	{attribute 'TcIecLibraryType'}
	{attribute 'external_name' := 'F_VN_CalibrateLinescanCameraExp_GUID_4678BC8A_FAF5_BD22_52B3_D89A3D1569BD'}
	(* Compute the camera parameters (intrinsic + extrinsic) by evaluating images containing a line calibration pattern. The pattern must consist of alternating vertical and diagonal lines, with each diagonal having the same constant slope: |\|\|...\|. The results are only valid for the x-direction of a line scan image. To get accurate x-values for a transformation into world coordinates, the y-coordinate must be set to half the sensor width and so equal to the cy-value of the camera matrix. For other y-values, the results are approximated and can be inaccurate. The extrinsic parameters are computed for the first image in the array. (expert function) *)
	FUNCTION F_VN_CalibrateLinescanCameraExp : HRESULT
	VAR_INPUT
		pSrcImages	:	PVOID;	(* Pointer to an array of 1 or more source images (1 channel). If the images have more than 1 row, each row must contain an image of the same pattern position. *)
		nSrcArraySize	:	UINT;	(* pSrcImages array size *)
		ipPatternLineOrigins	:	ITcVnContainer;	(* X position of the pattern line origins (ContainerType_Vector_REAL, usually same origin for vertical and following diagonal line) *)
		fSlopeRad	:	LREAL;	(* Slope of the diagonal line in rad (> 0, < PI/2), relative to the vertical line (i.e., 0 would be a vertical line, PI/2 a horizontal line) *)
	END_VAR
	VAR_IN_OUT
		aCameraMatrix	:	TcVnMatrix3x3_LREAL;	(* Returns the camera matrix *)
		aDistortionCoefficients	:	TcVnArray8_LREAL;	(* Returns the lens distortion coefficients [k1, k2, p1, p2, k3, k4, k5, k6] *)
		aRotationMatrix	:	TcVnMatrix3x3_LREAL;	(* Returns the rotation matrix *)
		aTranslationVector	:	TcVnVector3_LREAL;	(* Returns the translation vector *)
		fReprojError	:	LREAL;	(* Returns the reprojection error *)
		stCalibrationOptions	:	TcVnCameraCalibrationOptions;	(* Calibration options (recommended to set bFixAspectRatio, bFixPrincipalPoint, bZeroTangentDist) *)
	END_VAR
	VAR_INPUT
		eEdgeDirection	:	ETcVnEdgeDirection;	(* Specification of the edge direction to search for *)
		fMinStrength	:	REAL;	(* Specification of the minimum strength (intensity difference) of the edge to search for *)
		nMaxSearchLines	:	UDINT;	(* Maximum number of search lines (equally distributed over the image height, at most 1 searchline per image row) *)
		nMaxThickness	:	UDINT;	(* Specification of the maximum thickness of the edge to search for, which means fMinStrength must be reached within nMaxThickness pixels *)
		nSubpixelsIterations	:	UDINT;	(* Specifies the number of subpixels (for INTERPOLATION, 10 - 20 usually is sufficient) or maximum number of iterations for optimizing the parameters (for APPROX_ERF and APPROX_GAUSSIAN, 50 - 100 usually is sufficient) *)
		fApproxPrecision	:	REAL;	(* Specifies the approximation precision for APPROX_ERF and APPROX_GAUSSIAN (0.001 usually is sufficient, unused for INTERPOLATION) *)
		eAlgorithm	:	ETcVnEdgeDetectionAlgorithm;	(* Selection of the edge detection algorithm *)
		hrPrev	:	HRESULT;	(* HRESULT indicating the result of previous operations (If SUCCEEDED(hrPrev) equals false, no operation is executed.) *)
	END_VAR

END_FUNCTION

// Functions/Geometric and Coordinate Transformations/Calibration/F_VN_CompensateLensDistortion

	{attribute 'TcIecLibraryType'}
	{attribute 'external_name' := 'F_VN_CompensateLensDistortion_GUID_A3855505_9E36_B648_4D9A_72404444EE18'}
	(* Transforms an image to compensate the lens distortion. *)
	FUNCTION F_VN_CompensateLensDistortion : HRESULT
	VAR_INPUT
		ipSrcImage	:	ITcVnImage;	(* Source image *)
		ipDestImage	:	REFERENCE TO ITcVnImage;	(* Destination image (An appropriate destination image will be created if required.) *)
	END_VAR
	VAR_IN_OUT
		aCameraMatrix	:	TcVnMatrix3x3_LREAL;	(* Camera matrix containing the intrinsic parameters *)
		aDistortionCoefficients	:	TcVnArray4_LREAL;	(* Lens distortion coefficients [k1, k2, p1, p2] *)
	END_VAR
	VAR_INPUT
		hrPrev	:	HRESULT;	(* HRESULT indicating the result of previous operations (If SUCCEEDED(hrPrev) equals false, no operation is executed.) *)
	END_VAR

END_FUNCTION

// Functions/Geometric and Coordinate Transformations/Calibration/F_VN_CompensateLensDistortionExp1

	{attribute 'TcIecLibraryType'}
	{attribute 'external_name' := 'F_VN_CompensateLensDistortionExp1_GUID_39F83302_C215_BA53_4A0E_6585051CD298'}
	(* Transforms an image to compensate the lens distortion. (expert function) *)
	FUNCTION F_VN_CompensateLensDistortionExp1 : HRESULT
	VAR_INPUT
		ipSrcImage	:	ITcVnImage;	(* Source image *)
		ipDestImage	:	REFERENCE TO ITcVnImage;	(* Destination image (An appropriate destination image will be created if required.) *)
	END_VAR
	VAR_IN_OUT
		aCameraMatrix	:	TcVnMatrix3x3_LREAL;	(* Camera matrix containing the intrinsic parameters *)
		aDistortionCoefficients	:	TcVnArray8_LREAL;	(* Lens distortion coefficients [k1, k2, p1, p2, k3, k4, k5, k6] *)
	END_VAR
	VAR_INPUT
		hrPrev	:	HRESULT;	(* HRESULT indicating the result of previous operations (If SUCCEEDED(hrPrev) equals false, no operation is executed.) *)
	END_VAR

END_FUNCTION

// Functions/Geometric and Coordinate Transformations/Calibration/F_VN_CompensateLensDistortionExp2

	{attribute 'TcIecLibraryType'}
	{attribute 'external_name' := 'F_VN_CompensateLensDistortionExp2_GUID_C6636C8E_8710_BA51_6E0A_CA8278B52EE8'}
	(* Transforms an image to compensate the lens distortion. (expert function) *)
	FUNCTION F_VN_CompensateLensDistortionExp2 : HRESULT
	VAR_INPUT
		ipSrcImage	:	ITcVnImage;	(* Source image *)
		ipDestImage	:	REFERENCE TO ITcVnImage;	(* Destination image (An appropriate destination image will be created if required.) *)
	END_VAR
	VAR_IN_OUT
		aCameraMatrix	:	TcVnMatrix3x3_LREAL;	(* Camera matrix containing the intrinsic parameters *)
		aDistortionCoefficients	:	TcVnArray8_LREAL;	(* Lens distortion coefficients [k1, k2, p1, p2, k3, k4, k5, k6] *)
		aNewCameraMatrix	:	TcVnMatrix3x3_LREAL;	(* Allows additional scaling and shifting of the result image *)
	END_VAR
	VAR_INPUT
		hrPrev	:	HRESULT;	(* HRESULT indicating the result of previous operations (If SUCCEEDED(hrPrev) equals false, no operation is executed.) *)
	END_VAR

END_FUNCTION

// Functions/Geometric and Coordinate Transformations/Calibration/F_VN_CompensateLensDistortionForPoints

	{attribute 'TcIecLibraryType'}
	{attribute 'external_name' := 'F_VN_CompensateLensDistortionForPoints_GUID_1E1DEE69_79BC_BA65_762B_E597A5CC1182'}
	(* Transforms point coordinates to compensate the lens distortion. *)
	FUNCTION F_VN_CompensateLensDistortionForPoints : HRESULT
	VAR_INPUT
		ipSrcPoints	:	ITcVnContainer;	(* Container with source point coordinates (ContainerType_Vector_TcVnPoint2_REAL or ContainerType_Vector_TcVnPoint2_DINT) *)
		ipDestPoints	:	REFERENCE TO ITcVnContainer;	(* Returns a container with the transformed point coordinates (ContainerType_Vector_TcVnPoint2_REAL) *)
	END_VAR
	VAR_IN_OUT
		aCameraMatrix	:	TcVnMatrix3x3_LREAL;	(* Camera matrix containing the intrinsic parameters *)
		aDistortionCoefficients	:	TcVnArray4_LREAL;	(* Lens distortion coefficients [k1, k2, p1, p2] *)
	END_VAR
	VAR_INPUT
		hrPrev	:	HRESULT;	(* HRESULT indicating the result of previous operations (If SUCCEEDED(hrPrev) equals false, no operation is executed.) *)
	END_VAR

END_FUNCTION

// Functions/Geometric and Coordinate Transformations/Calibration/F_VN_CompensateLensDistortionForPointsExp1

	{attribute 'TcIecLibraryType'}
	{attribute 'external_name' := 'F_VN_CompensateLensDistortionForPointsExp1_GUID_7FE839DD_7A8B_BA4D_4709_CA0E7CDDBA0C'}
	(* Transforms point coordinates to compensate the lens distortion. (expert function) *)
	FUNCTION F_VN_CompensateLensDistortionForPointsExp1 : HRESULT
	VAR_INPUT
		ipSrcPoints	:	ITcVnContainer;	(* Container with source point coordinates (ContainerType_Vector_TcVnPoint2_REAL or ContainerType_Vector_TcVnPoint2_DINT) *)
		ipDestPoints	:	REFERENCE TO ITcVnContainer;	(* Returns a container with the transformed point coordinates (ContainerType_Vector_TcVnPoint2_REAL) *)
	END_VAR
	VAR_IN_OUT
		aCameraMatrix	:	TcVnMatrix3x3_LREAL;	(* Camera matrix containing the intrinsic parameters *)
		aDistortionCoefficients	:	TcVnArray8_LREAL;	(* Lens distortion coefficients [k1, k2, p1, p2, k3, k4, k5, k6] *)
	END_VAR
	VAR_INPUT
		hrPrev	:	HRESULT;	(* HRESULT indicating the result of previous operations (If SUCCEEDED(hrPrev) equals false, no operation is executed.) *)
	END_VAR

END_FUNCTION

// Functions/Geometric and Coordinate Transformations/Calibration/F_VN_CompensateLensDistortionForPointsExp2

	{attribute 'TcIecLibraryType'}
	{attribute 'external_name' := 'F_VN_CompensateLensDistortionForPointsExp2_GUID_30396D32_CFFC_B079_658D_44A89CF24BD9'}
	(* Transforms point coordinates to compensate the lens distortion. (expert function) *)
	FUNCTION F_VN_CompensateLensDistortionForPointsExp2 : HRESULT
	VAR_INPUT
		ipSrcPoints	:	ITcVnContainer;	(* Container with source point coordinates (ContainerType_Vector_TcVnPoint2_REAL or ContainerType_Vector_TcVnPoint2_DINT) *)
		ipDestPoints	:	REFERENCE TO ITcVnContainer;	(* Returns a container with the transformed point coordinates (ContainerType_Vector_TcVnPoint2_REAL) *)
	END_VAR
	VAR_IN_OUT
		aCameraMatrix	:	TcVnMatrix3x3_LREAL;	(* Camera matrix containing the intrinsic parameters *)
		aDistortionCoefficients	:	TcVnArray8_LREAL;	(* Lens distortion coefficients [k1, k2, p1, p2, k3, k4, k5, k6] *)
		aNewCameraMatrix	:	TcVnMatrix3x3_LREAL;	(* Allows additional shifting of the result point coordinates *)
	END_VAR
	VAR_INPUT
		hrPrev	:	HRESULT;	(* HRESULT indicating the result of previous operations (If SUCCEEDED(hrPrev) equals false, no operation is executed.) *)
	END_VAR

END_FUNCTION

// Functions/Geometric and Coordinate Transformations/Calibration/F_VN_DetectPatternPoints

	{attribute 'TcIecLibraryType'}
	{attribute 'external_name' := 'F_VN_DetectPatternPoints_GUID_E5D619D4_AB2C_BCDF_69FA_59048593E7EE'}
	(* Detects calibration pattern points (circles) within the provided image. *)
	FUNCTION F_VN_DetectPatternPoints : HRESULT
	VAR_INPUT
		ipSrcImage	:	ITcVnImage;	(* Source image (USINT, 1 channel) *)
		ipPatternPoints	:	REFERENCE TO ITcVnContainer;	(* Returns the pattern point positions (ContainerType_Vector_TcVnPoint2_REAL; Non-zero interface pointers are reused.) *)
	END_VAR
	VAR_IN_OUT
		stBlobDetectionParams	:	TcVnParamsBlobDetection;	(* Parameters to detect and filter contours. *)
	END_VAR
	VAR_INPUT
		nNumberOfPoints	:	UDINT;	(* Expected number of pattern points *)
		hrPrev	:	HRESULT;	(* HRESULT indicating the result of previous operations (If SUCCEEDED(hrPrev) equals false, no operation is executed.) *)
	END_VAR

END_FUNCTION

// Functions/Geometric and Coordinate Transformations/Calibration/F_VN_DetectPatternPointsExp

	{attribute 'TcIecLibraryType'}
	{attribute 'external_name' := 'F_VN_DetectPatternPointsExp_GUID_0BB96264_CC62_B28E_7E33_4178D5E9C206'}
	(* Detects calibration pattern points (circles) within the provided image. (expert function) *)
	FUNCTION F_VN_DetectPatternPointsExp : HRESULT
	VAR_INPUT
		ipSrcImage	:	ITcVnImage;	(* Source image (USINT, 1 channel) *)
		ipPatternPoints	:	REFERENCE TO ITcVnContainer;	(* Returns the pattern point positions (ContainerType_Vector_TcVnPoint2_REAL; Non-zero interface pointers are reused.) *)
	END_VAR
	VAR_IN_OUT
		stBlobDetectionParams	:	TcVnParamsBlobDetection;	(* Parameters to detect and filter contours. *)
	END_VAR
	VAR_INPUT
		nNumberOfPoints	:	UDINT;	(* Expected number of pattern points *)
		fSizeDiffThresFactor	:	REAL;	(* Threshold for filtering contours by average size *)
		bSubpixelAccuracy	:	BOOL;	(* If true, the pattern points are detected with subpixel accuracy *)
		eEdgeDirection	:	ETcVnEdgeDirection;	(* Specification of the edge direction to search for (from center to outside circle) *)
		fMinStrength	:	REAL;	(* Specification of the minimum strength (intensity difference) of the edge to search for *)
		nMaxThickness	:	UDINT;	(* Specification of the maximum thickness of the edge to search for, which means fMinStrength must be reached within nMaxThickness pixels *)
		nSubpixelsIterations	:	UDINT;	(* Specifies the number of subpixels (for INTERPOLATION, 10 - 20 usually is sufficient) or maximum number of iterations for optimizing the parameters (for APPROX_ERF and APPROX_GAUSSIAN, 50 - 100 usually is sufficient) *)
		nSearchLines	:	UDINT;	(* Specifies the amount of search lines, which are equally distributed in all directions (must be >= 8 and a multiple of 4) *)
		fApproxPrecision	:	REAL;	(* Specifies the approximation precision for APPROX_ERF and APPROX_GAUSSIAN (0.001 usually is sufficient, unused for INTERPOLATION) *)
		eAlgorithm	:	ETcVnEdgeDetectionAlgorithm;	(* Selection of the edge detection algorithm *)
		hrPrev	:	HRESULT;	(* HRESULT indicating the result of previous operations (If SUCCEEDED(hrPrev) equals false, no operation is executed.) *)
	END_VAR

END_FUNCTION

// Functions/Geometric and Coordinate Transformations/Calibration/F_VN_GenerateCalibrationPatternReferencePoints

	{attribute 'TcIecLibraryType'}
	{attribute 'external_name' := 'F_VN_GenerateCalibrationPatternReferencePoints_GUID_5DF6613C_109B_B749_6271_34E8C372E5AF'}
	(* Generate reference points for common calibration patterns. *)
	FUNCTION F_VN_GenerateCalibrationPatternReferencePoints : HRESULT
	VAR_INPUT
		ipReferencePoints	:	REFERENCE TO ITcVnContainer;	(* Returns the generated reference points (ContainerType_Vector_TcVnPoint3_REAL) *)
		ePattern	:	ETcVnCalibrationPattern;	(* Calibration pattern type *)
		eOrigin	:	ETcVnCalibrationPatternOrigin;	(* Calibration pattern origin *)
		nWidth	:	UDINT;	(* Pattern width, i.e. number of pattern points in x direction *)
		nHeight	:	UDINT;	(* Pattern height, i.e. number of pattern points in y direction *)
		fDistX	:	REAL;	(* Distance between pattern points in x direction *)
		fDistY	:	REAL;	(* Distance between pattern points in y direction *)
		hrPrev	:	HRESULT;	(* HRESULT indicating the result of previous operations (If SUCCEEDED(hrPrev) equals false, no operation is executed.) *)
	END_VAR

END_FUNCTION

// Functions/Geometric and Coordinate Transformations/Calibration/F_VN_ImagePointsWorldDistance

	{attribute 'TcIecLibraryType'}
	{attribute 'external_name' := 'F_VN_ImagePointsWorldDistance_GUID_0334DE15_3002_BBBB_566C_908DCC0EEAF4'}
	(* Computes the distance in the world coordinate system between two points (in the same world coordinate z layer) given in image coordinates. *)
	FUNCTION F_VN_ImagePointsWorldDistance : HRESULT
	VAR_IN_OUT
		aImagePoint1	:	TcVnPoint2_REAL;	(* First point in the image coordinate system *)
		aImagePoint2	:	TcVnPoint2_REAL;	(* Second point in the image coordinate system *)
		fWorldDistance	:	LREAL;	(* Returns the distance between aImagePoint1 and aImagePoint2 in the world coordinate system *)
		aCameraMatrix	:	TcVnMatrix3x3_LREAL;	(* 3x3 camera matrix containing the intrinsic parameters *)
		aDistortionCoefficients	:	TcVnArray8_LREAL;	(* Lens distortion coefficients [k1, k2, p1, p2, k3, k4, k5, k6] *)
		aRotationMatrix	:	TcVnMatrix3x3_LREAL;	(* 3x3 rotation matrix *)
		aTranslationVector	:	TcVnVector3_LREAL;	(* Translation vector *)
	END_VAR
	VAR_INPUT
		fZ	:	LREAL;	(* z coordinate (world coordinate system) of the given points (0 would be at (toplevel) calibration pattern) *)
		hrPrev	:	HRESULT;	(* HRESULT indicating the result of previous operations (If SUCCEEDED(hrPrev) equals false, no operation is executed.) *)
	END_VAR

END_FUNCTION

// Functions/Geometric and Coordinate Transformations/Calibration/F_VN_SolvePnP

	{attribute 'TcIecLibraryType'}
	{attribute 'external_name' := 'F_VN_SolvePnP_GUID_48B21731_B904_B5F9_506D_5F2F869F7C46'}
	(* Computes the rotation matrix and translation vector from 3D-2D point correspondences. *)
	FUNCTION F_VN_SolvePnP : HRESULT
	VAR_INPUT
		ipImagePoints	:	ITcVnContainer;	(* Image points (ContainerType_Vector_TcVnPoint2_REAL, requires at least 4 points in the same order as in ipReferencePoints) *)
		ipReferencePoints	:	ITcVnContainer;	(* Reference world points (ContainerType_Vector_TcVnPoint3_REAL, same number of points as in ipImagePoints) *)
	END_VAR
	VAR_IN_OUT
		aCameraMatrix	:	TcVnMatrix3x3_LREAL;	(* Camera matrix (e.g. computed with one of the CalibrateCamera functions) *)
		aDistortionCoefficients	:	TcVnArray8_LREAL;	(* Lens distortion coefficients [k1, k2, p1, p2, k3, k4, k5, k6] (e.g. computed with one of the CalibrateCamera functions) *)
		aRotationMatrix	:	TcVnMatrix3x3_LREAL;	(* Returns the rotation matrix *)
		aTranslationVector	:	TcVnVector3_LREAL;	(* Returns the translation vector *)
		fReprojError	:	LREAL;	(* Returns the reprojection error *)
	END_VAR
	VAR_INPUT
		hrPrev	:	HRESULT;	(* HRESULT indicating the result of previous operations (If SUCCEEDED(hrPrev) equals false, no operation is executed.) *)
	END_VAR

END_FUNCTION

// Functions/Geometric and Coordinate Transformations/Calibration/F_VN_SolvePnPExp

	{attribute 'TcIecLibraryType'}
	{attribute 'external_name' := 'F_VN_SolvePnPExp_GUID_4A6B57C8_30C5_B78E_7E73_5BBFD366FDC1'}
	(* Computes the rotation matrix and translation vector from 3D-2D point correspondences. (expert function) *)
	FUNCTION F_VN_SolvePnPExp : HRESULT
	VAR_INPUT
		ipImagePoints	:	ITcVnContainer;	(* Image points (ContainerType_Vector_TcVnPoint2_REAL, requires at least 4 points in the same order as in ipReferencePoints) *)
		ipReferencePoints	:	ITcVnContainer;	(* Reference world points (ContainerType_Vector_TcVnPoint3_REAL, same number of points as in ipImagePoints) *)
	END_VAR
	VAR_IN_OUT
		aCameraMatrix	:	TcVnMatrix3x3_LREAL;	(* Camera matrix (e.g. computed with one of the CalibrateCamera functions) *)
		aDistortionCoefficients	:	TcVnArray8_LREAL;	(* Lens distortion coefficients [k1, k2, p1, p2, k3, k4, k5, k6] (e.g. computed with one of the CalibrateCamera functions) *)
		aRotationMatrix	:	TcVnMatrix3x3_LREAL;	(* Returns the rotation matrix *)
		aTranslationVector	:	TcVnVector3_LREAL;	(* Returns the translation vector *)
		fReprojError	:	LREAL;	(* Returns the reprojection error *)
	END_VAR
	VAR_INPUT
		eMethod	:	ETcVnSolvePnPMethod;	(* Solve PnP method *)
		bUseExtrinsicGuess	:	BOOL;	(* If true, the provided rotation matrix and translation vector are used as an initial guess for further optimization (only supported for the SPM_ITERATIVE method). *)
		hrPrev	:	HRESULT;	(* HRESULT indicating the result of previous operations (If SUCCEEDED(hrPrev) equals false, no operation is executed.) *)
	END_VAR

END_FUNCTION

// Functions/Geometric and Coordinate Transformations/Calibration/F_VN_SortDetectedPatternPoints

	{attribute 'TcIecLibraryType'}
	{attribute 'external_name' := 'F_VN_SortDetectedPatternPoints_GUID_A17F6A56_659C_B437_7B82_7687D6CCA2D5'}
	(* Sort the detected pattern points according to the relative positions of the calibration pattern points. *)
	FUNCTION F_VN_SortDetectedPatternPoints : HRESULT
	VAR_INPUT
		ipImagePoints	:	ITcVnContainer;	(* Detected pattern point positions in the image coordinate system (will be sorted by this function, ContainerType_Vector_TcVnPoint2_REAL) *)
		ipPatternPoints	:	ITcVnContainer;	(* The pattern points in the calibration pattern coordinate system, used as a reference to sort ipImagePoints (ContainerType_Vector_TcVnPoint3_REAL) *)
		hrPrev	:	HRESULT;	(* HRESULT indicating the result of previous operations (If SUCCEEDED(hrPrev) equals false, no operation is executed.) *)
	END_VAR

END_FUNCTION

// Functions/Geometric and Coordinate Transformations/Calibration/F_VN_TransformCoordinatesPlanar_Container

	{attribute 'TcIecLibraryType'}
	{attribute 'external_name' := 'F_VN_TransformCoordinatesPlanar_Container_GUID_63387C97_18FC_B134_5620_A62F4E43774D'}
	(* Compute real-world coordinates for given image points or vice versa. *)
	FUNCTION F_VN_TransformCoordinatesPlanar_Container : HRESULT
	VAR_INPUT
		ipSrcPoints	:	ITcVnContainer;	(* Container with 2D source points (TcVnPoint2_DINT or TcVnPoint2_REAL or TcVnPoint2_LREAL) *)
		ipDestPoints	:	REFERENCE TO ITcVnContainer;	(* Returns the transformed 2D points (TcVnPoint2_LREAL) *)
	END_VAR
	VAR_IN_OUT
		aTransformationMatrix	:	TcVnMatrix3x3_LREAL;	(* Transformation matrix obtained with VnCalibrateCameraPlanar() or its inverse matrix obtained with VnInvertMatrix3x3() *)
	END_VAR
	VAR_INPUT
		hrPrev	:	HRESULT;	(* HRESULT indicating the result of previous operations (If SUCCEEDED(hrPrev) equals false, no operation is executed.) *)
	END_VAR

END_FUNCTION

// Functions/Geometric and Coordinate Transformations/Calibration/F_VN_TransformCoordinatesPlanar_Point

	{attribute 'TcIecLibraryType'}
	{attribute 'external_name' := 'F_VN_TransformCoordinatesPlanar_Point_GUID_97C2C18B_370F_B2DE_58FC_77BD7A1CF6B7'}
	(* Compute real-world coordinates for a given image point or vice versa. *)
	FUNCTION F_VN_TransformCoordinatesPlanar_Point : HRESULT
	VAR_IN_OUT
		aSrcPoint	:	TcVnPoint2_LREAL;	(* Point in the source coordinate system *)
		aDestPoint	:	TcVnPoint2_LREAL;	(* Returns point in the destination coordinate system *)
		aTransformationMatrix	:	TcVnMatrix3x3_LREAL;	(* Transformation matrix obtained with VnCalibrateCameraPlanar() or its inverse matrix obtained with VnInvertMatrix3x3() *)
	END_VAR
	VAR_INPUT
		hrPrev	:	HRESULT;	(* HRESULT indicating the result of previous operations (If SUCCEEDED(hrPrev) equals false, no operation is executed.) *)
	END_VAR

END_FUNCTION

// Functions/Geometric and Coordinate Transformations/Calibration/F_VN_TransformCoordinatesImageToWorld_Container

	{attribute 'TcIecLibraryType'}
	{attribute 'external_name' := 'F_VN_TransformCoordinatesImageToWorld_Container_GUID_50AFD962_6C8A_B091_690A_6E7AB7BA8507'}
	(* Transform 2D image point coordinates to 3D world coordinates (using intrinsic + extrinsic calibration results). *)
	FUNCTION F_VN_TransformCoordinatesImageToWorld_Container : HRESULT
	VAR_INPUT
		ipSrcPoints2D	:	ITcVnContainer;	(* Container with 2D source points (TcVnPoint2_DINT or TcVnPoint2_REAL or TcVnPoint2_LREAL) *)
		ipDestPoints3D	:	REFERENCE TO ITcVnContainer;	(* Returns the transformed 3D points (TcVnPoint3_LREAL) *)
	END_VAR
	VAR_IN_OUT
		aCameraMatrix	:	TcVnMatrix3x3_LREAL;	(* 3x3 camera matrix containing the intrinsic parameters *)
		aDistortionCoefficients	:	TcVnArray8_LREAL;	(* Lens distortion coefficients [k1, k2, p1, p2, k3, k4, k5, k6] *)
		aRotationMatrix	:	TcVnMatrix3x3_LREAL;	(* 3x3 rotation matrix *)
		aTranslationVector	:	TcVnVector3_LREAL;	(* Translation vector *)
	END_VAR
	VAR_INPUT
		fZ	:	LREAL;	(* z coordinate (world coordinate system) of the transformed points (0 would be at (toplevel) calibration pattern) *)
		hrPrev	:	HRESULT;	(* HRESULT indicating the result of previous operations (If SUCCEEDED(hrPrev) equals false, no operation is executed.) *)
	END_VAR

END_FUNCTION

// Functions/Geometric and Coordinate Transformations/Calibration/F_VN_TransformCoordinatesImageToWorld_Point

	{attribute 'TcIecLibraryType'}
	{attribute 'external_name' := 'F_VN_TransformCoordinatesImageToWorld_Point_GUID_878D3094_5879_B155_5FE7_7FEE3864E859'}
	(* Transform 2D image point coordinate to 3D world coordinate (using intrinsic + extrinsic calibration results). *)
	FUNCTION F_VN_TransformCoordinatesImageToWorld_Point : HRESULT
	VAR_IN_OUT
		aSrcPoint	:	TcVnPoint2_LREAL;	(* Point in the image coordinate system *)
		aDestPoint	:	TcVnPoint3_LREAL;	(* Returns the point in the world coordinate system *)
		aCameraMatrix	:	TcVnMatrix3x3_LREAL;	(* 3x3 camera matrix containing the intrinsic parameters *)
		aDistortionCoefficients	:	TcVnArray8_LREAL;	(* Lens distortion coefficients [k1, k2, p1, p2, k3, k4, k5, k6] *)
		aRotationMatrix	:	TcVnMatrix3x3_LREAL;	(* 3x3 rotation matrix *)
		aTranslationVector	:	TcVnVector3_LREAL;	(* Translation vector *)
	END_VAR
	VAR_INPUT
		fZ	:	LREAL;	(* z coordinate (world coordinate system) of the transformed points (0 would be at (toplevel) calibration pattern) *)
		hrPrev	:	HRESULT;	(* HRESULT indicating the result of previous operations (If SUCCEEDED(hrPrev) equals false, no operation is executed.) *)
	END_VAR

END_FUNCTION

// Functions/Geometric and Coordinate Transformations/Calibration/F_VN_TransformCoordinatesWorldToImage_Container

	{attribute 'TcIecLibraryType'}
	{attribute 'external_name' := 'F_VN_TransformCoordinatesWorldToImage_Container_GUID_C2B9C466_778A_BF1D_5F76_D14708CB6927'}
	(* Transform 3D world coordinates to 2D image coordinates (using intrinsic + extrinsic calibration results). *)
	FUNCTION F_VN_TransformCoordinatesWorldToImage_Container : HRESULT
	VAR_INPUT
		ipSrcPoints3D	:	ITcVnContainer;	(* Container with 3D source points (TcVnPoint3_LREAL) *)
		ipDestPoints2D	:	REFERENCE TO ITcVnContainer;	(* Returns the transformed 2D points (TcVnPoint2_REAL or TcVnPoint2_DINT, depending on bInteger) *)
	END_VAR
	VAR_IN_OUT
		aCameraMatrix	:	TcVnMatrix3x3_LREAL;	(* 3x3 camera matrix containing the intrinsic parameters *)
		aDistortionCoefficients	:	TcVnArray8_LREAL;	(* Lens distortion coefficients [k1, k2, p1, p2, k3, k4, k5, k6] *)
		aRotationMatrix	:	TcVnMatrix3x3_LREAL;	(* 3x3 rotation matrix *)
		aTranslationVector	:	TcVnVector3_LREAL;	(* Translation vector *)
	END_VAR
	VAR_INPUT
		bInteger	:	BOOL;	(* Selects whether the function returns a container of TcVnPoint2_DINT or TcVnPoint2_REAL *)
		hrPrev	:	HRESULT;	(* HRESULT indicating the result of previous operations (If SUCCEEDED(hrPrev) equals false, no operation is executed.) *)
	END_VAR

END_FUNCTION

// Functions/Geometric and Coordinate Transformations/Calibration/F_VN_TransformCoordinatesWorldToImage_Point

	{attribute 'TcIecLibraryType'}
	{attribute 'external_name' := 'F_VN_TransformCoordinatesWorldToImage_Point_GUID_868BAD46_546E_B47F_5D29_201948E8ED29'}
	(* Transform 3D world coordinates to 2D image coordinates (using intrinsic + extrinsic calibration results). *)
	FUNCTION F_VN_TransformCoordinatesWorldToImage_Point : HRESULT
	VAR_IN_OUT
		aSrcPoint	:	TcVnPoint3_LREAL;	(* 3D source point (world coordinate system) *)
		aDestPoint	:	TcVnPoint2_REAL;	(* Returns the transformed 2D point (image coordinate system) *)
		aCameraMatrix	:	TcVnMatrix3x3_LREAL;	(* 3x3 camera matrix containing the intrinsic parameters *)
		aDistortionCoefficients	:	TcVnArray8_LREAL;	(* Lens distortion coefficients [k1, k2, p1, p2, k3, k4, k5, k6] *)
		aRotationMatrix	:	TcVnMatrix3x3_LREAL;	(* 3x3 rotation matrix *)
		aTranslationVector	:	TcVnVector3_LREAL;	(* Translation vector *)
	END_VAR
	VAR_INPUT
		hrPrev	:	HRESULT;	(* HRESULT indicating the result of previous operations (If SUCCEEDED(hrPrev) equals false, no operation is executed.) *)
	END_VAR

END_FUNCTION

// Functions/Container Statistics/F_VN_MaxElementElementwise/F_VN_MaxElementElementwise_DINT

	{attribute 'TcIecLibraryType'}
	{attribute 'external_name' := 'F_VN_MaxElementElementwise_DINT_GUID_A1BE4267_BA1B_BA90_67BB_3DBFC1859A8F'}
	(* Gets the element wise maximum container element. *)
	FUNCTION F_VN_MaxElementElementwise_DINT : HRESULT
	VAR_INPUT
		ipContainer	:	ITcVnContainer;	(* Source container *)
	END_VAR
	VAR_IN_OUT
		nMax	:	DINT;	(* Returns the requested element *)
	END_VAR
	VAR_INPUT
		hrPrev	:	HRESULT;	(* HRESULT indicating the result of previous operations (If SUCCEEDED(hrPrev) equals false, no operation is executed.) *)
	END_VAR

END_FUNCTION

// Functions/Container Statistics/F_VN_MaxElementElementwise/F_VN_MaxElementElementwise_INT

	{attribute 'TcIecLibraryType'}
	{attribute 'external_name' := 'F_VN_MaxElementElementwise_INT_GUID_95B7CFD0_0FD8_B93B_5C5E_7D47F827E85F'}
	(* Gets the element wise maximum container element. *)
	FUNCTION F_VN_MaxElementElementwise_INT : HRESULT
	VAR_INPUT
		ipContainer	:	ITcVnContainer;	(* Source container *)
	END_VAR
	VAR_IN_OUT
		nMax	:	INT;	(* Returns the requested element *)
	END_VAR
	VAR_INPUT
		hrPrev	:	HRESULT;	(* HRESULT indicating the result of previous operations (If SUCCEEDED(hrPrev) equals false, no operation is executed.) *)
	END_VAR

END_FUNCTION

// Functions/Container Statistics/F_VN_MaxElementElementwise/F_VN_MaxElementElementwise_LREAL

	{attribute 'TcIecLibraryType'}
	{attribute 'external_name' := 'F_VN_MaxElementElementwise_LREAL_GUID_420A3B04_1DFF_B5FC_5DCD_BC08562F4A21'}
	(* Gets the element wise maximum container element. *)
	FUNCTION F_VN_MaxElementElementwise_LREAL : HRESULT
	VAR_INPUT
		ipContainer	:	ITcVnContainer;	(* Source container *)
	END_VAR
	VAR_IN_OUT
		fMax	:	LREAL;	(* Returns the requested element *)
	END_VAR
	VAR_INPUT
		hrPrev	:	HRESULT;	(* HRESULT indicating the result of previous operations (If SUCCEEDED(hrPrev) equals false, no operation is executed.) *)
	END_VAR

END_FUNCTION

// Functions/Container Statistics/F_VN_MaxElementElementwise/F_VN_MaxElementElementwise_REAL

	{attribute 'TcIecLibraryType'}
	{attribute 'external_name' := 'F_VN_MaxElementElementwise_REAL_GUID_29FB8FF1_899E_B8DF_50CD_57BBD70290AF'}
	(* Gets the element wise maximum container element. *)
	FUNCTION F_VN_MaxElementElementwise_REAL : HRESULT
	VAR_INPUT
		ipContainer	:	ITcVnContainer;	(* Source container *)
	END_VAR
	VAR_IN_OUT
		fMax	:	REAL;	(* Returns the requested element *)
	END_VAR
	VAR_INPUT
		hrPrev	:	HRESULT;	(* HRESULT indicating the result of previous operations (If SUCCEEDED(hrPrev) equals false, no operation is executed.) *)
	END_VAR

END_FUNCTION

// Functions/Container Statistics/F_VN_MaxElementElementwise/F_VN_MaxElementElementwise_SINT

	{attribute 'TcIecLibraryType'}
	{attribute 'external_name' := 'F_VN_MaxElementElementwise_SINT_GUID_D76AA4A4_55AC_B7D3_77EE_1A3750AFA155'}
	(* Gets the element wise maximum container element. *)
	FUNCTION F_VN_MaxElementElementwise_SINT : HRESULT
	VAR_INPUT
		ipContainer	:	ITcVnContainer;	(* Source container *)
	END_VAR
	VAR_IN_OUT
		nMax	:	SINT;	(* Returns the requested element *)
	END_VAR
	VAR_INPUT
		hrPrev	:	HRESULT;	(* HRESULT indicating the result of previous operations (If SUCCEEDED(hrPrev) equals false, no operation is executed.) *)
	END_VAR

END_FUNCTION

// Functions/Container Statistics/F_VN_MaxElementElementwise/F_VN_MaxElementElementwise_TcVnPoint2_DINT

	{attribute 'TcIecLibraryType'}
	{attribute 'external_name' := 'F_VN_MaxElementElementwise_TcVnPoint2_DINT_GUID_AB8D48FE_9E5C_BBD1_45E8_F5959AC4978C'}
	(* Gets the element wise maximum container element. *)
	FUNCTION F_VN_MaxElementElementwise_TcVnPoint2_DINT : HRESULT
	VAR_INPUT
		ipContainer	:	ITcVnContainer;	(* Source container *)
	END_VAR
	VAR_IN_OUT
		aMax	:	TcVnPoint2_DINT;	(* Returns the requested element *)
	END_VAR
	VAR_INPUT
		hrPrev	:	HRESULT;	(* HRESULT indicating the result of previous operations (If SUCCEEDED(hrPrev) equals false, no operation is executed.) *)
	END_VAR

END_FUNCTION

// Functions/Container Statistics/F_VN_MaxElementElementwise/F_VN_MaxElementElementwise_TcVnPoint2_LREAL

	{attribute 'TcIecLibraryType'}
	{attribute 'external_name' := 'F_VN_MaxElementElementwise_TcVnPoint2_LREAL_GUID_A5ED05D2_D29F_BB40_609E_53217FDA123C'}
	(* Gets the element wise maximum container element. *)
	FUNCTION F_VN_MaxElementElementwise_TcVnPoint2_LREAL : HRESULT
	VAR_INPUT
		ipContainer	:	ITcVnContainer;	(* Source container *)
	END_VAR
	VAR_IN_OUT
		aMax	:	TcVnPoint2_LREAL;	(* Returns the requested element *)
	END_VAR
	VAR_INPUT
		hrPrev	:	HRESULT;	(* HRESULT indicating the result of previous operations (If SUCCEEDED(hrPrev) equals false, no operation is executed.) *)
	END_VAR

END_FUNCTION

// Functions/Container Statistics/F_VN_MaxElementElementwise/F_VN_MaxElementElementwise_TcVnPoint2_REAL

	{attribute 'TcIecLibraryType'}
	{attribute 'external_name' := 'F_VN_MaxElementElementwise_TcVnPoint2_REAL_GUID_0E1407D4_05E1_B824_4214_30F3E2475EA8'}
	(* Gets the element wise maximum container element. *)
	FUNCTION F_VN_MaxElementElementwise_TcVnPoint2_REAL : HRESULT
	VAR_INPUT
		ipContainer	:	ITcVnContainer;	(* Source container *)
	END_VAR
	VAR_IN_OUT
		aMax	:	TcVnPoint2_REAL;	(* Returns the requested element *)
	END_VAR
	VAR_INPUT
		hrPrev	:	HRESULT;	(* HRESULT indicating the result of previous operations (If SUCCEEDED(hrPrev) equals false, no operation is executed.) *)
	END_VAR

END_FUNCTION

// Functions/Container Statistics/F_VN_MaxElementElementwise/F_VN_MaxElementElementwise_TcVnPoint3_LREAL

	{attribute 'TcIecLibraryType'}
	{attribute 'external_name' := 'F_VN_MaxElementElementwise_TcVnPoint3_LREAL_GUID_0A41620C_B32E_B639_6154_C38E83DCF80E'}
	(* Gets the element wise maximum container element. *)
	FUNCTION F_VN_MaxElementElementwise_TcVnPoint3_LREAL : HRESULT
	VAR_INPUT
		ipContainer	:	ITcVnContainer;	(* Source container *)
	END_VAR
	VAR_IN_OUT
		aMax	:	TcVnPoint3_LREAL;	(* Returns the requested element *)
	END_VAR
	VAR_INPUT
		hrPrev	:	HRESULT;	(* HRESULT indicating the result of previous operations (If SUCCEEDED(hrPrev) equals false, no operation is executed.) *)
	END_VAR

END_FUNCTION

// Functions/Container Statistics/F_VN_MaxElementElementwise/F_VN_MaxElementElementwise_TcVnPoint3_REAL

	{attribute 'TcIecLibraryType'}
	{attribute 'external_name' := 'F_VN_MaxElementElementwise_TcVnPoint3_REAL_GUID_FD9C75FE_2428_B795_667F_E3F06A1869C3'}
	(* Gets the element wise maximum container element. *)
	FUNCTION F_VN_MaxElementElementwise_TcVnPoint3_REAL : HRESULT
	VAR_INPUT
		ipContainer	:	ITcVnContainer;	(* Source container *)
	END_VAR
	VAR_IN_OUT
		aMax	:	TcVnPoint3_REAL;	(* Returns the requested element *)
	END_VAR
	VAR_INPUT
		hrPrev	:	HRESULT;	(* HRESULT indicating the result of previous operations (If SUCCEEDED(hrPrev) equals false, no operation is executed.) *)
	END_VAR

END_FUNCTION

// Functions/Container Statistics/F_VN_MaxElementElementwise/F_VN_MaxElementElementwise_TcVnVector2_DINT

	{attribute 'TcIecLibraryType'}
	{attribute 'external_name' := 'F_VN_MaxElementElementwise_TcVnVector2_DINT_GUID_C3E2FECF_4970_B1DE_76C8_1A94F4358646'}
	(* Gets the element wise maximum container element. *)
	FUNCTION F_VN_MaxElementElementwise_TcVnVector2_DINT : HRESULT
	VAR_INPUT
		ipContainer	:	ITcVnContainer;	(* Source container *)
	END_VAR
	VAR_IN_OUT
		aMax	:	TcVnVector2_DINT;	(* Returns the requested element *)
	END_VAR
	VAR_INPUT
		hrPrev	:	HRESULT;	(* HRESULT indicating the result of previous operations (If SUCCEEDED(hrPrev) equals false, no operation is executed.) *)
	END_VAR

END_FUNCTION

// Functions/Container Statistics/F_VN_MaxElementElementwise/F_VN_MaxElementElementwise_TcVnVector2_INT

	{attribute 'TcIecLibraryType'}
	{attribute 'external_name' := 'F_VN_MaxElementElementwise_TcVnVector2_INT_GUID_CA6DB23B_1F56_BB53_6A44_9B9E6F523DD6'}
	(* Gets the element wise maximum container element. *)
	FUNCTION F_VN_MaxElementElementwise_TcVnVector2_INT : HRESULT
	VAR_INPUT
		ipContainer	:	ITcVnContainer;	(* Source container *)
	END_VAR
	VAR_IN_OUT
		aMax	:	TcVnVector2_INT;	(* Returns the requested element *)
	END_VAR
	VAR_INPUT
		hrPrev	:	HRESULT;	(* HRESULT indicating the result of previous operations (If SUCCEEDED(hrPrev) equals false, no operation is executed.) *)
	END_VAR

END_FUNCTION

// Functions/Container Statistics/F_VN_MaxElementElementwise/F_VN_MaxElementElementwise_TcVnVector2_REAL

	{attribute 'TcIecLibraryType'}
	{attribute 'external_name' := 'F_VN_MaxElementElementwise_TcVnVector2_REAL_GUID_AD7ED1D9_ACC6_BD18_7659_4390CA2823BD'}
	(* Gets the element wise maximum container element. *)
	FUNCTION F_VN_MaxElementElementwise_TcVnVector2_REAL : HRESULT
	VAR_INPUT
		ipContainer	:	ITcVnContainer;	(* Source container *)
	END_VAR
	VAR_IN_OUT
		aMax	:	TcVnVector2_REAL;	(* Returns the requested element *)
	END_VAR
	VAR_INPUT
		hrPrev	:	HRESULT;	(* HRESULT indicating the result of previous operations (If SUCCEEDED(hrPrev) equals false, no operation is executed.) *)
	END_VAR

END_FUNCTION

// Functions/Container Statistics/F_VN_MaxElementElementwise/F_VN_MaxElementElementwise_TcVnVector2_SINT

	{attribute 'TcIecLibraryType'}
	{attribute 'external_name' := 'F_VN_MaxElementElementwise_TcVnVector2_SINT_GUID_29A36FC3_DA56_B072_501D_7F8D455A6F7E'}
	(* Gets the element wise maximum container element. *)
	FUNCTION F_VN_MaxElementElementwise_TcVnVector2_SINT : HRESULT
	VAR_INPUT
		ipContainer	:	ITcVnContainer;	(* Source container *)
	END_VAR
	VAR_IN_OUT
		aMax	:	TcVnVector2_SINT;	(* Returns the requested element *)
	END_VAR
	VAR_INPUT
		hrPrev	:	HRESULT;	(* HRESULT indicating the result of previous operations (If SUCCEEDED(hrPrev) equals false, no operation is executed.) *)
	END_VAR

END_FUNCTION

// Functions/Container Statistics/F_VN_MaxElementElementwise/F_VN_MaxElementElementwise_TcVnVector2_UINT

	{attribute 'TcIecLibraryType'}
	{attribute 'external_name' := 'F_VN_MaxElementElementwise_TcVnVector2_UINT_GUID_BB7E8C0D_7764_BA5C_51E9_69D403A67F7A'}
	(* Gets the element wise maximum container element. *)
	FUNCTION F_VN_MaxElementElementwise_TcVnVector2_UINT : HRESULT
	VAR_INPUT
		ipContainer	:	ITcVnContainer;	(* Source container *)
	END_VAR
	VAR_IN_OUT
		aMax	:	TcVnVector2_UINT;	(* Returns the requested element *)
	END_VAR
	VAR_INPUT
		hrPrev	:	HRESULT;	(* HRESULT indicating the result of previous operations (If SUCCEEDED(hrPrev) equals false, no operation is executed.) *)
	END_VAR

END_FUNCTION

// Functions/Container Statistics/F_VN_MaxElementElementwise/F_VN_MaxElementElementwise_TcVnVector2_USINT

	{attribute 'TcIecLibraryType'}
	{attribute 'external_name' := 'F_VN_MaxElementElementwise_TcVnVector2_USINT_GUID_EE16444C_FD5F_BC7B_50DF_F5A4C4ED6E17'}
	(* Gets the element wise maximum container element. *)
	FUNCTION F_VN_MaxElementElementwise_TcVnVector2_USINT : HRESULT
	VAR_INPUT
		ipContainer	:	ITcVnContainer;	(* Source container *)
	END_VAR
	VAR_IN_OUT
		aMax	:	TcVnVector2_USINT;	(* Returns the requested element *)
	END_VAR
	VAR_INPUT
		hrPrev	:	HRESULT;	(* HRESULT indicating the result of previous operations (If SUCCEEDED(hrPrev) equals false, no operation is executed.) *)
	END_VAR

END_FUNCTION

// Functions/Container Statistics/F_VN_MaxElementElementwise/F_VN_MaxElementElementwise_TcVnVector3_INT

	{attribute 'TcIecLibraryType'}
	{attribute 'external_name' := 'F_VN_MaxElementElementwise_TcVnVector3_INT_GUID_1980FFD2_2EAF_B070_4ED3_E9AA766C9471'}
	(* Gets the element wise maximum container element. *)
	FUNCTION F_VN_MaxElementElementwise_TcVnVector3_INT : HRESULT
	VAR_INPUT
		ipContainer	:	ITcVnContainer;	(* Source container *)
	END_VAR
	VAR_IN_OUT
		aMax	:	TcVnVector3_INT;	(* Returns the requested element *)
	END_VAR
	VAR_INPUT
		hrPrev	:	HRESULT;	(* HRESULT indicating the result of previous operations (If SUCCEEDED(hrPrev) equals false, no operation is executed.) *)
	END_VAR

END_FUNCTION

// Functions/Container Statistics/F_VN_MaxElementElementwise/F_VN_MaxElementElementwise_TcVnVector3_REAL

	{attribute 'TcIecLibraryType'}
	{attribute 'external_name' := 'F_VN_MaxElementElementwise_TcVnVector3_REAL_GUID_9A360533_8CF8_BC7C_45B7_3BD6F1E36E2D'}
	(* Gets the element wise maximum container element. *)
	FUNCTION F_VN_MaxElementElementwise_TcVnVector3_REAL : HRESULT
	VAR_INPUT
		ipContainer	:	ITcVnContainer;	(* Source container *)
	END_VAR
	VAR_IN_OUT
		aMax	:	TcVnVector3_REAL;	(* Returns the requested element *)
	END_VAR
	VAR_INPUT
		hrPrev	:	HRESULT;	(* HRESULT indicating the result of previous operations (If SUCCEEDED(hrPrev) equals false, no operation is executed.) *)
	END_VAR

END_FUNCTION

// Functions/Container Statistics/F_VN_MaxElementElementwise/F_VN_MaxElementElementwise_TcVnVector3_SINT

	{attribute 'TcIecLibraryType'}
	{attribute 'external_name' := 'F_VN_MaxElementElementwise_TcVnVector3_SINT_GUID_F97DE7EC_9F07_BD75_51B0_2EEF81C4D76B'}
	(* Gets the element wise maximum container element. *)
	FUNCTION F_VN_MaxElementElementwise_TcVnVector3_SINT : HRESULT
	VAR_INPUT
		ipContainer	:	ITcVnContainer;	(* Source container *)
	END_VAR
	VAR_IN_OUT
		aMax	:	TcVnVector3_SINT;	(* Returns the requested element *)
	END_VAR
	VAR_INPUT
		hrPrev	:	HRESULT;	(* HRESULT indicating the result of previous operations (If SUCCEEDED(hrPrev) equals false, no operation is executed.) *)
	END_VAR

END_FUNCTION

// Functions/Container Statistics/F_VN_MaxElementElementwise/F_VN_MaxElementElementwise_TcVnVector3_UINT

	{attribute 'TcIecLibraryType'}
	{attribute 'external_name' := 'F_VN_MaxElementElementwise_TcVnVector3_UINT_GUID_8C4B741F_8652_B04F_7E59_9F73B5BD6B17'}
	(* Gets the element wise maximum container element. *)
	FUNCTION F_VN_MaxElementElementwise_TcVnVector3_UINT : HRESULT
	VAR_INPUT
		ipContainer	:	ITcVnContainer;	(* Source container *)
	END_VAR
	VAR_IN_OUT
		aMax	:	TcVnVector3_UINT;	(* Returns the requested element *)
	END_VAR
	VAR_INPUT
		hrPrev	:	HRESULT;	(* HRESULT indicating the result of previous operations (If SUCCEEDED(hrPrev) equals false, no operation is executed.) *)
	END_VAR

END_FUNCTION

// Functions/Container Statistics/F_VN_MaxElementElementwise/F_VN_MaxElementElementwise_TcVnVector3_USINT

	{attribute 'TcIecLibraryType'}
	{attribute 'external_name' := 'F_VN_MaxElementElementwise_TcVnVector3_USINT_GUID_51CB88E5_EA47_BEC4_4D37_CE48B0966640'}
	(* Gets the element wise maximum container element. *)
	FUNCTION F_VN_MaxElementElementwise_TcVnVector3_USINT : HRESULT
	VAR_INPUT
		ipContainer	:	ITcVnContainer;	(* Source container *)
	END_VAR
	VAR_IN_OUT
		aMax	:	TcVnVector3_USINT;	(* Returns the requested element *)
	END_VAR
	VAR_INPUT
		hrPrev	:	HRESULT;	(* HRESULT indicating the result of previous operations (If SUCCEEDED(hrPrev) equals false, no operation is executed.) *)
	END_VAR

END_FUNCTION

// Functions/Container Statistics/F_VN_MaxElementElementwise/F_VN_MaxElementElementwise_TcVnVector4_DINT

	{attribute 'TcIecLibraryType'}
	{attribute 'external_name' := 'F_VN_MaxElementElementwise_TcVnVector4_DINT_GUID_56B3CAC2_02B4_B5A4_6BA7_9B69A08F2962'}
	(* Gets the element wise maximum container element. *)
	FUNCTION F_VN_MaxElementElementwise_TcVnVector4_DINT : HRESULT
	VAR_INPUT
		ipContainer	:	ITcVnContainer;	(* Source container *)
	END_VAR
	VAR_IN_OUT
		aMax	:	TcVnVector4_DINT;	(* Returns the requested element *)
	END_VAR
	VAR_INPUT
		hrPrev	:	HRESULT;	(* HRESULT indicating the result of previous operations (If SUCCEEDED(hrPrev) equals false, no operation is executed.) *)
	END_VAR

END_FUNCTION

// Functions/Container Statistics/F_VN_MaxElementElementwise/F_VN_MaxElementElementwise_TcVnVector4_INT

	{attribute 'TcIecLibraryType'}
	{attribute 'external_name' := 'F_VN_MaxElementElementwise_TcVnVector4_INT_GUID_84A706B7_0C05_B7A5_5565_3FA88BAD6F2D'}
	(* Gets the element wise maximum container element. *)
	FUNCTION F_VN_MaxElementElementwise_TcVnVector4_INT : HRESULT
	VAR_INPUT
		ipContainer	:	ITcVnContainer;	(* Source container *)
	END_VAR
	VAR_IN_OUT
		aMax	:	TcVnVector4_INT;	(* Returns the requested element *)
	END_VAR
	VAR_INPUT
		hrPrev	:	HRESULT;	(* HRESULT indicating the result of previous operations (If SUCCEEDED(hrPrev) equals false, no operation is executed.) *)
	END_VAR

END_FUNCTION

// Functions/Container Statistics/F_VN_MaxElementElementwise/F_VN_MaxElementElementwise_TcVnVector4_LREAL

	{attribute 'TcIecLibraryType'}
	{attribute 'external_name' := 'F_VN_MaxElementElementwise_TcVnVector4_LREAL_GUID_6C873FDB_D55C_BABB_5D7C_28C50FA85179'}
	(* Gets the element wise maximum container element. *)
	FUNCTION F_VN_MaxElementElementwise_TcVnVector4_LREAL : HRESULT
	VAR_INPUT
		ipContainer	:	ITcVnContainer;	(* Source container *)
	END_VAR
	VAR_IN_OUT
		aMax	:	TcVnVector4_LREAL;	(* Returns the requested element *)
	END_VAR
	VAR_INPUT
		hrPrev	:	HRESULT;	(* HRESULT indicating the result of previous operations (If SUCCEEDED(hrPrev) equals false, no operation is executed.) *)
	END_VAR

END_FUNCTION

// Functions/Container Statistics/F_VN_MaxElementElementwise/F_VN_MaxElementElementwise_TcVnVector4_SINT

	{attribute 'TcIecLibraryType'}
	{attribute 'external_name' := 'F_VN_MaxElementElementwise_TcVnVector4_SINT_GUID_2036C25B_5973_B0A1_4A2E_82AC57D81D5C'}
	(* Gets the element wise maximum container element. *)
	FUNCTION F_VN_MaxElementElementwise_TcVnVector4_SINT : HRESULT
	VAR_INPUT
		ipContainer	:	ITcVnContainer;	(* Source container *)
	END_VAR
	VAR_IN_OUT
		aMax	:	TcVnVector4_SINT;	(* Returns the requested element *)
	END_VAR
	VAR_INPUT
		hrPrev	:	HRESULT;	(* HRESULT indicating the result of previous operations (If SUCCEEDED(hrPrev) equals false, no operation is executed.) *)
	END_VAR

END_FUNCTION

// Functions/Container Statistics/F_VN_MaxElementElementwise/F_VN_MaxElementElementwise_TcVnVector4_UINT

	{attribute 'TcIecLibraryType'}
	{attribute 'external_name' := 'F_VN_MaxElementElementwise_TcVnVector4_UINT_GUID_FE6C3D2B_7298_BD2F_5599_4CA9627F2B97'}
	(* Gets the element wise maximum container element. *)
	FUNCTION F_VN_MaxElementElementwise_TcVnVector4_UINT : HRESULT
	VAR_INPUT
		ipContainer	:	ITcVnContainer;	(* Source container *)
	END_VAR
	VAR_IN_OUT
		aMax	:	TcVnVector4_UINT;	(* Returns the requested element *)
	END_VAR
	VAR_INPUT
		hrPrev	:	HRESULT;	(* HRESULT indicating the result of previous operations (If SUCCEEDED(hrPrev) equals false, no operation is executed.) *)
	END_VAR

END_FUNCTION

// Functions/Container Statistics/F_VN_MaxElementElementwise/F_VN_MaxElementElementwise_TcVnVector4_USINT

	{attribute 'TcIecLibraryType'}
	{attribute 'external_name' := 'F_VN_MaxElementElementwise_TcVnVector4_USINT_GUID_07B5E611_A95A_B7DD_74B8_4C3EFE7A1E88'}
	(* Gets the element wise maximum container element. *)
	FUNCTION F_VN_MaxElementElementwise_TcVnVector4_USINT : HRESULT
	VAR_INPUT
		ipContainer	:	ITcVnContainer;	(* Source container *)
	END_VAR
	VAR_IN_OUT
		aMax	:	TcVnVector4_USINT;	(* Returns the requested element *)
	END_VAR
	VAR_INPUT
		hrPrev	:	HRESULT;	(* HRESULT indicating the result of previous operations (If SUCCEEDED(hrPrev) equals false, no operation is executed.) *)
	END_VAR

END_FUNCTION

// Functions/Container Statistics/F_VN_MaxElementElementwise/F_VN_MaxElementElementwise_UDINT

	{attribute 'TcIecLibraryType'}
	{attribute 'external_name' := 'F_VN_MaxElementElementwise_UDINT_GUID_B4CACA11_92FF_BE6E_46F5_2138F457FA4F'}
	(* Gets the element wise maximum container element. *)
	FUNCTION F_VN_MaxElementElementwise_UDINT : HRESULT
	VAR_INPUT
		ipContainer	:	ITcVnContainer;	(* Source container *)
	END_VAR
	VAR_IN_OUT
		nMax	:	UDINT;	(* Returns the requested element *)
	END_VAR
	VAR_INPUT
		hrPrev	:	HRESULT;	(* HRESULT indicating the result of previous operations (If SUCCEEDED(hrPrev) equals false, no operation is executed.) *)
	END_VAR

END_FUNCTION

// Functions/Container Statistics/F_VN_MaxElementElementwise/F_VN_MaxElementElementwise_UINT

	{attribute 'TcIecLibraryType'}
	{attribute 'external_name' := 'F_VN_MaxElementElementwise_UINT_GUID_B704428E_BF70_BDF8_60BC_D91087754694'}
	(* Gets the element wise maximum container element. *)
	FUNCTION F_VN_MaxElementElementwise_UINT : HRESULT
	VAR_INPUT
		ipContainer	:	ITcVnContainer;	(* Source container *)
	END_VAR
	VAR_IN_OUT
		nMax	:	UINT;	(* Returns the requested element *)
	END_VAR
	VAR_INPUT
		hrPrev	:	HRESULT;	(* HRESULT indicating the result of previous operations (If SUCCEEDED(hrPrev) equals false, no operation is executed.) *)
	END_VAR

END_FUNCTION

// Functions/Container Statistics/F_VN_MaxElementElementwise/F_VN_MaxElementElementwise_ULINT

	{attribute 'TcIecLibraryType'}
	{attribute 'external_name' := 'F_VN_MaxElementElementwise_ULINT_GUID_E2D6111D_3D44_BAA0_4CA2_782393F5EB39'}
	(* Gets the element wise maximum container element. *)
	FUNCTION F_VN_MaxElementElementwise_ULINT : HRESULT
	VAR_INPUT
		ipContainer	:	ITcVnContainer;	(* Source container *)
	END_VAR
	VAR_IN_OUT
		nMax	:	ULINT;	(* Returns the requested element *)
	END_VAR
	VAR_INPUT
		hrPrev	:	HRESULT;	(* HRESULT indicating the result of previous operations (If SUCCEEDED(hrPrev) equals false, no operation is executed.) *)
	END_VAR

END_FUNCTION

// Functions/Container Statistics/F_VN_MaxElementElementwise/F_VN_MaxElementElementwise_USINT

	{attribute 'TcIecLibraryType'}
	{attribute 'external_name' := 'F_VN_MaxElementElementwise_USINT_GUID_FE64BC6C_1A07_BE42_5CF4_5D54DFD4400D'}
	(* Gets the element wise maximum container element. *)
	FUNCTION F_VN_MaxElementElementwise_USINT : HRESULT
	VAR_INPUT
		ipContainer	:	ITcVnContainer;	(* Source container *)
	END_VAR
	VAR_IN_OUT
		nMax	:	USINT;	(* Returns the requested element *)
	END_VAR
	VAR_INPUT
		hrPrev	:	HRESULT;	(* HRESULT indicating the result of previous operations (If SUCCEEDED(hrPrev) equals false, no operation is executed.) *)
	END_VAR

END_FUNCTION

// Functions/Container Statistics/F_VN_MedianElementElementwise/F_VN_MedianElementElementwise_DINT

	{attribute 'TcIecLibraryType'}
	{attribute 'external_name' := 'F_VN_MedianElementElementwise_DINT_GUID_B22BC711_B45B_BCC1_57C1_06B1120E9F4C'}
	(* Gets the element wise median container element. *)
	FUNCTION F_VN_MedianElementElementwise_DINT : HRESULT
	VAR_INPUT
		ipContainer	:	ITcVnContainer;	(* Source container *)
	END_VAR
	VAR_IN_OUT
		nMedian	:	DINT;	(* Returns the requested element *)
	END_VAR
	VAR_INPUT
		hrPrev	:	HRESULT;	(* HRESULT indicating the result of previous operations (If SUCCEEDED(hrPrev) equals false, no operation is executed.) *)
	END_VAR

END_FUNCTION

// Functions/Container Statistics/F_VN_MedianElementElementwise/F_VN_MedianElementElementwise_INT

	{attribute 'TcIecLibraryType'}
	{attribute 'external_name' := 'F_VN_MedianElementElementwise_INT_GUID_508B8619_B3FA_B9CA_5BEB_AA72C8BFDF3D'}
	(* Gets the element wise median container element. *)
	FUNCTION F_VN_MedianElementElementwise_INT : HRESULT
	VAR_INPUT
		ipContainer	:	ITcVnContainer;	(* Source container *)
	END_VAR
	VAR_IN_OUT
		nMedian	:	INT;	(* Returns the requested element *)
	END_VAR
	VAR_INPUT
		hrPrev	:	HRESULT;	(* HRESULT indicating the result of previous operations (If SUCCEEDED(hrPrev) equals false, no operation is executed.) *)
	END_VAR

END_FUNCTION

// Functions/Container Statistics/F_VN_MedianElementElementwise/F_VN_MedianElementElementwise_LREAL

	{attribute 'TcIecLibraryType'}
	{attribute 'external_name' := 'F_VN_MedianElementElementwise_LREAL_GUID_2EE05F32_CBF3_B774_74A9_CD6E359092B0'}
	(* Gets the element wise median container element. *)
	FUNCTION F_VN_MedianElementElementwise_LREAL : HRESULT
	VAR_INPUT
		ipContainer	:	ITcVnContainer;	(* Source container *)
	END_VAR
	VAR_IN_OUT
		fMedian	:	LREAL;	(* Returns the requested element *)
	END_VAR
	VAR_INPUT
		hrPrev	:	HRESULT;	(* HRESULT indicating the result of previous operations (If SUCCEEDED(hrPrev) equals false, no operation is executed.) *)
	END_VAR

END_FUNCTION

// Functions/Container Statistics/F_VN_MedianElementElementwise/F_VN_MedianElementElementwise_REAL

	{attribute 'TcIecLibraryType'}
	{attribute 'external_name' := 'F_VN_MedianElementElementwise_REAL_GUID_BA5FB88A_CFF2_B702_5385_5BB60F0279F8'}
	(* Gets the element wise median container element. *)
	FUNCTION F_VN_MedianElementElementwise_REAL : HRESULT
	VAR_INPUT
		ipContainer	:	ITcVnContainer;	(* Source container *)
	END_VAR
	VAR_IN_OUT
		fMedian	:	REAL;	(* Returns the requested element *)
	END_VAR
	VAR_INPUT
		hrPrev	:	HRESULT;	(* HRESULT indicating the result of previous operations (If SUCCEEDED(hrPrev) equals false, no operation is executed.) *)
	END_VAR

END_FUNCTION

// Functions/Container Statistics/F_VN_MedianElementElementwise/F_VN_MedianElementElementwise_SINT

	{attribute 'TcIecLibraryType'}
	{attribute 'external_name' := 'F_VN_MedianElementElementwise_SINT_GUID_3CEA1FEB_55B1_B380_7E49_AF86F63A8D16'}
	(* Gets the element wise median container element. *)
	FUNCTION F_VN_MedianElementElementwise_SINT : HRESULT
	VAR_INPUT
		ipContainer	:	ITcVnContainer;	(* Source container *)
	END_VAR
	VAR_IN_OUT
		nMedian	:	SINT;	(* Returns the requested element *)
	END_VAR
	VAR_INPUT
		hrPrev	:	HRESULT;	(* HRESULT indicating the result of previous operations (If SUCCEEDED(hrPrev) equals false, no operation is executed.) *)
	END_VAR

END_FUNCTION

// Functions/Container Statistics/F_VN_MedianElementElementwise/F_VN_MedianElementElementwise_TcVnPoint2_DINT

	{attribute 'TcIecLibraryType'}
	{attribute 'external_name' := 'F_VN_MedianElementElementwise_TcVnPoint2_DINT_GUID_38D86DE0_157C_BC4B_5BA9_BF8EC0C0027B'}
	(* Gets the element wise median container element. *)
	FUNCTION F_VN_MedianElementElementwise_TcVnPoint2_DINT : HRESULT
	VAR_INPUT
		ipContainer	:	ITcVnContainer;	(* Source container *)
	END_VAR
	VAR_IN_OUT
		aMedian	:	TcVnPoint2_DINT;	(* Returns the requested element *)
	END_VAR
	VAR_INPUT
		hrPrev	:	HRESULT;	(* HRESULT indicating the result of previous operations (If SUCCEEDED(hrPrev) equals false, no operation is executed.) *)
	END_VAR

END_FUNCTION

// Functions/Container Statistics/F_VN_MedianElementElementwise/F_VN_MedianElementElementwise_TcVnPoint2_LREAL

	{attribute 'TcIecLibraryType'}
	{attribute 'external_name' := 'F_VN_MedianElementElementwise_TcVnPoint2_LREAL_GUID_C32B8676_0BD7_BBCE_420D_3A61654B88A9'}
	(* Gets the element wise median container element. *)
	FUNCTION F_VN_MedianElementElementwise_TcVnPoint2_LREAL : HRESULT
	VAR_INPUT
		ipContainer	:	ITcVnContainer;	(* Source container *)
	END_VAR
	VAR_IN_OUT
		aMedian	:	TcVnPoint2_LREAL;	(* Returns the requested element *)
	END_VAR
	VAR_INPUT
		hrPrev	:	HRESULT;	(* HRESULT indicating the result of previous operations (If SUCCEEDED(hrPrev) equals false, no operation is executed.) *)
	END_VAR

END_FUNCTION

// Functions/Container Statistics/F_VN_MedianElementElementwise/F_VN_MedianElementElementwise_TcVnPoint2_REAL

	{attribute 'TcIecLibraryType'}
	{attribute 'external_name' := 'F_VN_MedianElementElementwise_TcVnPoint2_REAL_GUID_63D2322B_784A_B21B_7139_73FFA1E949A9'}
	(* Gets the element wise median container element. *)
	FUNCTION F_VN_MedianElementElementwise_TcVnPoint2_REAL : HRESULT
	VAR_INPUT
		ipContainer	:	ITcVnContainer;	(* Source container *)
	END_VAR
	VAR_IN_OUT
		aMedian	:	TcVnPoint2_REAL;	(* Returns the requested element *)
	END_VAR
	VAR_INPUT
		hrPrev	:	HRESULT;	(* HRESULT indicating the result of previous operations (If SUCCEEDED(hrPrev) equals false, no operation is executed.) *)
	END_VAR

END_FUNCTION

// Functions/Container Statistics/F_VN_MedianElementElementwise/F_VN_MedianElementElementwise_TcVnPoint3_LREAL

	{attribute 'TcIecLibraryType'}
	{attribute 'external_name' := 'F_VN_MedianElementElementwise_TcVnPoint3_LREAL_GUID_6ACB7222_737C_BCA0_44EF_4FEB11884B22'}
	(* Gets the element wise median container element. *)
	FUNCTION F_VN_MedianElementElementwise_TcVnPoint3_LREAL : HRESULT
	VAR_INPUT
		ipContainer	:	ITcVnContainer;	(* Source container *)
	END_VAR
	VAR_IN_OUT
		aMedian	:	TcVnPoint3_LREAL;	(* Returns the requested element *)
	END_VAR
	VAR_INPUT
		hrPrev	:	HRESULT;	(* HRESULT indicating the result of previous operations (If SUCCEEDED(hrPrev) equals false, no operation is executed.) *)
	END_VAR

END_FUNCTION

// Functions/Container Statistics/F_VN_MedianElementElementwise/F_VN_MedianElementElementwise_TcVnPoint3_REAL

	{attribute 'TcIecLibraryType'}
	{attribute 'external_name' := 'F_VN_MedianElementElementwise_TcVnPoint3_REAL_GUID_EEEE6964_26F6_BF33_4B71_DB76D10F29D1'}
	(* Gets the element wise median container element. *)
	FUNCTION F_VN_MedianElementElementwise_TcVnPoint3_REAL : HRESULT
	VAR_INPUT
		ipContainer	:	ITcVnContainer;	(* Source container *)
	END_VAR
	VAR_IN_OUT
		aMedian	:	TcVnPoint3_REAL;	(* Returns the requested element *)
	END_VAR
	VAR_INPUT
		hrPrev	:	HRESULT;	(* HRESULT indicating the result of previous operations (If SUCCEEDED(hrPrev) equals false, no operation is executed.) *)
	END_VAR

END_FUNCTION

// Functions/Container Statistics/F_VN_MedianElementElementwise/F_VN_MedianElementElementwise_TcVnVector2_DINT

	{attribute 'TcIecLibraryType'}
	{attribute 'external_name' := 'F_VN_MedianElementElementwise_TcVnVector2_DINT_GUID_15C674BB_F6C5_BB69_76F5_3635732E6AC1'}
	(* Gets the element wise median container element. *)
	FUNCTION F_VN_MedianElementElementwise_TcVnVector2_DINT : HRESULT
	VAR_INPUT
		ipContainer	:	ITcVnContainer;	(* Source container *)
	END_VAR
	VAR_IN_OUT
		aMedian	:	TcVnVector2_DINT;	(* Returns the requested element *)
	END_VAR
	VAR_INPUT
		hrPrev	:	HRESULT;	(* HRESULT indicating the result of previous operations (If SUCCEEDED(hrPrev) equals false, no operation is executed.) *)
	END_VAR

END_FUNCTION

// Functions/Container Statistics/F_VN_MedianElementElementwise/F_VN_MedianElementElementwise_TcVnVector2_INT

	{attribute 'TcIecLibraryType'}
	{attribute 'external_name' := 'F_VN_MedianElementElementwise_TcVnVector2_INT_GUID_C05C75F2_E397_BA41_49DE_1D67A9E1ACEC'}
	(* Gets the element wise median container element. *)
	FUNCTION F_VN_MedianElementElementwise_TcVnVector2_INT : HRESULT
	VAR_INPUT
		ipContainer	:	ITcVnContainer;	(* Source container *)
	END_VAR
	VAR_IN_OUT
		aMedian	:	TcVnVector2_INT;	(* Returns the requested element *)
	END_VAR
	VAR_INPUT
		hrPrev	:	HRESULT;	(* HRESULT indicating the result of previous operations (If SUCCEEDED(hrPrev) equals false, no operation is executed.) *)
	END_VAR

END_FUNCTION

// Functions/Container Statistics/F_VN_MedianElementElementwise/F_VN_MedianElementElementwise_TcVnVector2_REAL

	{attribute 'TcIecLibraryType'}
	{attribute 'external_name' := 'F_VN_MedianElementElementwise_TcVnVector2_REAL_GUID_1D68FE03_B2F0_B3E5_7EBD_F59E16CA8C63'}
	(* Gets the element wise median container element. *)
	FUNCTION F_VN_MedianElementElementwise_TcVnVector2_REAL : HRESULT
	VAR_INPUT
		ipContainer	:	ITcVnContainer;	(* Source container *)
	END_VAR
	VAR_IN_OUT
		aMedian	:	TcVnVector2_REAL;	(* Returns the requested element *)
	END_VAR
	VAR_INPUT
		hrPrev	:	HRESULT;	(* HRESULT indicating the result of previous operations (If SUCCEEDED(hrPrev) equals false, no operation is executed.) *)
	END_VAR

END_FUNCTION

// Functions/Container Statistics/F_VN_MedianElementElementwise/F_VN_MedianElementElementwise_TcVnVector2_SINT

	{attribute 'TcIecLibraryType'}
	{attribute 'external_name' := 'F_VN_MedianElementElementwise_TcVnVector2_SINT_GUID_64A65886_F3B2_BB3F_6DE1_0163972635FE'}
	(* Gets the element wise median container element. *)
	FUNCTION F_VN_MedianElementElementwise_TcVnVector2_SINT : HRESULT
	VAR_INPUT
		ipContainer	:	ITcVnContainer;	(* Source container *)
	END_VAR
	VAR_IN_OUT
		aMedian	:	TcVnVector2_SINT;	(* Returns the requested element *)
	END_VAR
	VAR_INPUT
		hrPrev	:	HRESULT;	(* HRESULT indicating the result of previous operations (If SUCCEEDED(hrPrev) equals false, no operation is executed.) *)
	END_VAR

END_FUNCTION

// Functions/Container Statistics/F_VN_MedianElementElementwise/F_VN_MedianElementElementwise_TcVnVector2_UINT

	{attribute 'TcIecLibraryType'}
	{attribute 'external_name' := 'F_VN_MedianElementElementwise_TcVnVector2_UINT_GUID_EBD93672_2E86_B8F1_4134_F8DDF87340A8'}
	(* Gets the element wise median container element. *)
	FUNCTION F_VN_MedianElementElementwise_TcVnVector2_UINT : HRESULT
	VAR_INPUT
		ipContainer	:	ITcVnContainer;	(* Source container *)
	END_VAR
	VAR_IN_OUT
		aMedian	:	TcVnVector2_UINT;	(* Returns the requested element *)
	END_VAR
	VAR_INPUT
		hrPrev	:	HRESULT;	(* HRESULT indicating the result of previous operations (If SUCCEEDED(hrPrev) equals false, no operation is executed.) *)
	END_VAR

END_FUNCTION

// Functions/Container Statistics/F_VN_MedianElementElementwise/F_VN_MedianElementElementwise_TcVnVector2_USINT

	{attribute 'TcIecLibraryType'}
	{attribute 'external_name' := 'F_VN_MedianElementElementwise_TcVnVector2_USINT_GUID_BEF15B44_7427_B887_718C_FFCF0E78029C'}
	(* Gets the element wise median container element. *)
	FUNCTION F_VN_MedianElementElementwise_TcVnVector2_USINT : HRESULT
	VAR_INPUT
		ipContainer	:	ITcVnContainer;	(* Source container *)
	END_VAR
	VAR_IN_OUT
		aMedian	:	TcVnVector2_USINT;	(* Returns the requested element *)
	END_VAR
	VAR_INPUT
		hrPrev	:	HRESULT;	(* HRESULT indicating the result of previous operations (If SUCCEEDED(hrPrev) equals false, no operation is executed.) *)
	END_VAR

END_FUNCTION

// Functions/Container Statistics/F_VN_MedianElementElementwise/F_VN_MedianElementElementwise_TcVnVector3_INT

	{attribute 'TcIecLibraryType'}
	{attribute 'external_name' := 'F_VN_MedianElementElementwise_TcVnVector3_INT_GUID_D75797A2_A89E_B659_4391_5481F0584504'}
	(* Gets the element wise median container element. *)
	FUNCTION F_VN_MedianElementElementwise_TcVnVector3_INT : HRESULT
	VAR_INPUT
		ipContainer	:	ITcVnContainer;	(* Source container *)
	END_VAR
	VAR_IN_OUT
		aMedian	:	TcVnVector3_INT;	(* Returns the requested element *)
	END_VAR
	VAR_INPUT
		hrPrev	:	HRESULT;	(* HRESULT indicating the result of previous operations (If SUCCEEDED(hrPrev) equals false, no operation is executed.) *)
	END_VAR

END_FUNCTION

// Functions/Container Statistics/F_VN_MedianElementElementwise/F_VN_MedianElementElementwise_TcVnVector3_REAL

	{attribute 'TcIecLibraryType'}
	{attribute 'external_name' := 'F_VN_MedianElementElementwise_TcVnVector3_REAL_GUID_D5180C4A_88BE_BA94_7B81_B2395553BD8C'}
	(* Gets the element wise median container element. *)
	FUNCTION F_VN_MedianElementElementwise_TcVnVector3_REAL : HRESULT
	VAR_INPUT
		ipContainer	:	ITcVnContainer;	(* Source container *)
	END_VAR
	VAR_IN_OUT
		aMedian	:	TcVnVector3_REAL;	(* Returns the requested element *)
	END_VAR
	VAR_INPUT
		hrPrev	:	HRESULT;	(* HRESULT indicating the result of previous operations (If SUCCEEDED(hrPrev) equals false, no operation is executed.) *)
	END_VAR

END_FUNCTION

// Functions/Container Statistics/F_VN_MedianElementElementwise/F_VN_MedianElementElementwise_TcVnVector3_SINT

	{attribute 'TcIecLibraryType'}
	{attribute 'external_name' := 'F_VN_MedianElementElementwise_TcVnVector3_SINT_GUID_0AB6949C_5E21_B681_6D97_FCE689970370'}
	(* Gets the element wise median container element. *)
	FUNCTION F_VN_MedianElementElementwise_TcVnVector3_SINT : HRESULT
	VAR_INPUT
		ipContainer	:	ITcVnContainer;	(* Source container *)
	END_VAR
	VAR_IN_OUT
		aMedian	:	TcVnVector3_SINT;	(* Returns the requested element *)
	END_VAR
	VAR_INPUT
		hrPrev	:	HRESULT;	(* HRESULT indicating the result of previous operations (If SUCCEEDED(hrPrev) equals false, no operation is executed.) *)
	END_VAR

END_FUNCTION

// Functions/Container Statistics/F_VN_MedianElementElementwise/F_VN_MedianElementElementwise_TcVnVector3_UINT

	{attribute 'TcIecLibraryType'}
	{attribute 'external_name' := 'F_VN_MedianElementElementwise_TcVnVector3_UINT_GUID_335ECED1_1723_BC32_7DA0_4B01AE021AA4'}
	(* Gets the element wise median container element. *)
	FUNCTION F_VN_MedianElementElementwise_TcVnVector3_UINT : HRESULT
	VAR_INPUT
		ipContainer	:	ITcVnContainer;	(* Source container *)
	END_VAR
	VAR_IN_OUT
		aMedian	:	TcVnVector3_UINT;	(* Returns the requested element *)
	END_VAR
	VAR_INPUT
		hrPrev	:	HRESULT;	(* HRESULT indicating the result of previous operations (If SUCCEEDED(hrPrev) equals false, no operation is executed.) *)
	END_VAR

END_FUNCTION

// Functions/Container Statistics/F_VN_MedianElementElementwise/F_VN_MedianElementElementwise_TcVnVector3_USINT

	{attribute 'TcIecLibraryType'}
	{attribute 'external_name' := 'F_VN_MedianElementElementwise_TcVnVector3_USINT_GUID_970ED975_5A4F_B4DC_72E6_B00E212F06DE'}
	(* Gets the element wise median container element. *)
	FUNCTION F_VN_MedianElementElementwise_TcVnVector3_USINT : HRESULT
	VAR_INPUT
		ipContainer	:	ITcVnContainer;	(* Source container *)
	END_VAR
	VAR_IN_OUT
		aMedian	:	TcVnVector3_USINT;	(* Returns the requested element *)
	END_VAR
	VAR_INPUT
		hrPrev	:	HRESULT;	(* HRESULT indicating the result of previous operations (If SUCCEEDED(hrPrev) equals false, no operation is executed.) *)
	END_VAR

END_FUNCTION

// Functions/Container Statistics/F_VN_MedianElementElementwise/F_VN_MedianElementElementwise_TcVnVector4_DINT

	{attribute 'TcIecLibraryType'}
	{attribute 'external_name' := 'F_VN_MedianElementElementwise_TcVnVector4_DINT_GUID_F42CEA87_5060_B19A_78A3_D2D5E0B685B0'}
	(* Gets the element wise median container element. *)
	FUNCTION F_VN_MedianElementElementwise_TcVnVector4_DINT : HRESULT
	VAR_INPUT
		ipContainer	:	ITcVnContainer;	(* Source container *)
	END_VAR
	VAR_IN_OUT
		aMedian	:	TcVnVector4_DINT;	(* Returns the requested element *)
	END_VAR
	VAR_INPUT
		hrPrev	:	HRESULT;	(* HRESULT indicating the result of previous operations (If SUCCEEDED(hrPrev) equals false, no operation is executed.) *)
	END_VAR

END_FUNCTION

// Functions/Container Statistics/F_VN_MedianElementElementwise/F_VN_MedianElementElementwise_TcVnVector4_INT

	{attribute 'TcIecLibraryType'}
	{attribute 'external_name' := 'F_VN_MedianElementElementwise_TcVnVector4_INT_GUID_CFFAEC06_3E73_B9A1_6F3A_1C5FA22F88D8'}
	(* Gets the element wise median container element. *)
	FUNCTION F_VN_MedianElementElementwise_TcVnVector4_INT : HRESULT
	VAR_INPUT
		ipContainer	:	ITcVnContainer;	(* Source container *)
	END_VAR
	VAR_IN_OUT
		aMedian	:	TcVnVector4_INT;	(* Returns the requested element *)
	END_VAR
	VAR_INPUT
		hrPrev	:	HRESULT;	(* HRESULT indicating the result of previous operations (If SUCCEEDED(hrPrev) equals false, no operation is executed.) *)
	END_VAR

END_FUNCTION

// Functions/Container Statistics/F_VN_MedianElementElementwise/F_VN_MedianElementElementwise_TcVnVector4_LREAL

	{attribute 'TcIecLibraryType'}
	{attribute 'external_name' := 'F_VN_MedianElementElementwise_TcVnVector4_LREAL_GUID_F9E74369_0B03_BA15_47B9_5D4745B46A4D'}
	(* Gets the element wise median container element. *)
	FUNCTION F_VN_MedianElementElementwise_TcVnVector4_LREAL : HRESULT
	VAR_INPUT
		ipContainer	:	ITcVnContainer;	(* Source container *)
	END_VAR
	VAR_IN_OUT
		aMedian	:	TcVnVector4_LREAL;	(* Returns the requested element *)
	END_VAR
	VAR_INPUT
		hrPrev	:	HRESULT;	(* HRESULT indicating the result of previous operations (If SUCCEEDED(hrPrev) equals false, no operation is executed.) *)
	END_VAR

END_FUNCTION

// Functions/Container Statistics/F_VN_MedianElementElementwise/F_VN_MedianElementElementwise_TcVnVector4_SINT

	{attribute 'TcIecLibraryType'}
	{attribute 'external_name' := 'F_VN_MedianElementElementwise_TcVnVector4_SINT_GUID_FAE81295_409D_B7A6_6F19_D3F5AE675BEF'}
	(* Gets the element wise median container element. *)
	FUNCTION F_VN_MedianElementElementwise_TcVnVector4_SINT : HRESULT
	VAR_INPUT
		ipContainer	:	ITcVnContainer;	(* Source container *)
	END_VAR
	VAR_IN_OUT
		aMedian	:	TcVnVector4_SINT;	(* Returns the requested element *)
	END_VAR
	VAR_INPUT
		hrPrev	:	HRESULT;	(* HRESULT indicating the result of previous operations (If SUCCEEDED(hrPrev) equals false, no operation is executed.) *)
	END_VAR

END_FUNCTION

// Functions/Container Statistics/F_VN_MedianElementElementwise/F_VN_MedianElementElementwise_TcVnVector4_UINT

	{attribute 'TcIecLibraryType'}
	{attribute 'external_name' := 'F_VN_MedianElementElementwise_TcVnVector4_UINT_GUID_9F3CF28C_220F_B7DF_7AA7_69E81D701262'}
	(* Gets the element wise median container element. *)
	FUNCTION F_VN_MedianElementElementwise_TcVnVector4_UINT : HRESULT
	VAR_INPUT
		ipContainer	:	ITcVnContainer;	(* Source container *)
	END_VAR
	VAR_IN_OUT
		aMedian	:	TcVnVector4_UINT;	(* Returns the requested element *)
	END_VAR
	VAR_INPUT
		hrPrev	:	HRESULT;	(* HRESULT indicating the result of previous operations (If SUCCEEDED(hrPrev) equals false, no operation is executed.) *)
	END_VAR

END_FUNCTION

// Functions/Container Statistics/F_VN_MedianElementElementwise/F_VN_MedianElementElementwise_TcVnVector4_USINT

	{attribute 'TcIecLibraryType'}
	{attribute 'external_name' := 'F_VN_MedianElementElementwise_TcVnVector4_USINT_GUID_5D9344EE_1EC5_B92A_45E9_540F2094E30B'}
	(* Gets the element wise median container element. *)
	FUNCTION F_VN_MedianElementElementwise_TcVnVector4_USINT : HRESULT
	VAR_INPUT
		ipContainer	:	ITcVnContainer;	(* Source container *)
	END_VAR
	VAR_IN_OUT
		aMedian	:	TcVnVector4_USINT;	(* Returns the requested element *)
	END_VAR
	VAR_INPUT
		hrPrev	:	HRESULT;	(* HRESULT indicating the result of previous operations (If SUCCEEDED(hrPrev) equals false, no operation is executed.) *)
	END_VAR

END_FUNCTION

// Functions/Container Statistics/F_VN_MedianElementElementwise/F_VN_MedianElementElementwise_UDINT

	{attribute 'TcIecLibraryType'}
	{attribute 'external_name' := 'F_VN_MedianElementElementwise_UDINT_GUID_0046FE0C_602C_B383_7FC2_9A4C9D50B20D'}
	(* Gets the element wise median container element. *)
	FUNCTION F_VN_MedianElementElementwise_UDINT : HRESULT
	VAR_INPUT
		ipContainer	:	ITcVnContainer;	(* Source container *)
	END_VAR
	VAR_IN_OUT
		nMedian	:	UDINT;	(* Returns the requested element *)
	END_VAR
	VAR_INPUT
		hrPrev	:	HRESULT;	(* HRESULT indicating the result of previous operations (If SUCCEEDED(hrPrev) equals false, no operation is executed.) *)
	END_VAR

END_FUNCTION

// Functions/Container Statistics/F_VN_MedianElementElementwise/F_VN_MedianElementElementwise_UINT

	{attribute 'TcIecLibraryType'}
	{attribute 'external_name' := 'F_VN_MedianElementElementwise_UINT_GUID_31FF4568_76D4_B543_6111_6F4C3F3FD5F3'}
	(* Gets the element wise median container element. *)
	FUNCTION F_VN_MedianElementElementwise_UINT : HRESULT
	VAR_INPUT
		ipContainer	:	ITcVnContainer;	(* Source container *)
	END_VAR
	VAR_IN_OUT
		nMedian	:	UINT;	(* Returns the requested element *)
	END_VAR
	VAR_INPUT
		hrPrev	:	HRESULT;	(* HRESULT indicating the result of previous operations (If SUCCEEDED(hrPrev) equals false, no operation is executed.) *)
	END_VAR

END_FUNCTION

// Functions/Container Statistics/F_VN_MedianElementElementwise/F_VN_MedianElementElementwise_ULINT

	{attribute 'TcIecLibraryType'}
	{attribute 'external_name' := 'F_VN_MedianElementElementwise_ULINT_GUID_154EFE3B_5F4A_BE7B_4735_58FFBB2DFB6D'}
	(* Gets the element wise median container element. *)
	FUNCTION F_VN_MedianElementElementwise_ULINT : HRESULT
	VAR_INPUT
		ipContainer	:	ITcVnContainer;	(* Source container *)
	END_VAR
	VAR_IN_OUT
		nMedian	:	ULINT;	(* Returns the requested element *)
	END_VAR
	VAR_INPUT
		hrPrev	:	HRESULT;	(* HRESULT indicating the result of previous operations (If SUCCEEDED(hrPrev) equals false, no operation is executed.) *)
	END_VAR

END_FUNCTION

// Functions/Container Statistics/F_VN_MedianElementElementwise/F_VN_MedianElementElementwise_USINT

	{attribute 'TcIecLibraryType'}
	{attribute 'external_name' := 'F_VN_MedianElementElementwise_USINT_GUID_B215C911_D93A_BC50_52A9_FBE963CE6AEA'}
	(* Gets the element wise median container element. *)
	FUNCTION F_VN_MedianElementElementwise_USINT : HRESULT
	VAR_INPUT
		ipContainer	:	ITcVnContainer;	(* Source container *)
	END_VAR
	VAR_IN_OUT
		nMedian	:	USINT;	(* Returns the requested element *)
	END_VAR
	VAR_INPUT
		hrPrev	:	HRESULT;	(* HRESULT indicating the result of previous operations (If SUCCEEDED(hrPrev) equals false, no operation is executed.) *)
	END_VAR

END_FUNCTION

// Functions/Container Statistics/F_VN_MinElementElementwise/F_VN_MinElementElementwise_DINT

	{attribute 'TcIecLibraryType'}
	{attribute 'external_name' := 'F_VN_MinElementElementwise_DINT_GUID_E5D73089_CAD8_B7AF_6F7B_961D7517D0AD'}
	(* Gets the element wise minimum container element. *)
	FUNCTION F_VN_MinElementElementwise_DINT : HRESULT
	VAR_INPUT
		ipContainer	:	ITcVnContainer;	(* Source container *)
	END_VAR
	VAR_IN_OUT
		nMin	:	DINT;	(* Returns the requested element *)
	END_VAR
	VAR_INPUT
		hrPrev	:	HRESULT;	(* HRESULT indicating the result of previous operations (If SUCCEEDED(hrPrev) equals false, no operation is executed.) *)
	END_VAR

END_FUNCTION

// Functions/Container Statistics/F_VN_MinElementElementwise/F_VN_MinElementElementwise_INT

	{attribute 'TcIecLibraryType'}
	{attribute 'external_name' := 'F_VN_MinElementElementwise_INT_GUID_90381010_37C5_B5BF_5FEF_FBDB48C10B30'}
	(* Gets the element wise minimum container element. *)
	FUNCTION F_VN_MinElementElementwise_INT : HRESULT
	VAR_INPUT
		ipContainer	:	ITcVnContainer;	(* Source container *)
	END_VAR
	VAR_IN_OUT
		nMin	:	INT;	(* Returns the requested element *)
	END_VAR
	VAR_INPUT
		hrPrev	:	HRESULT;	(* HRESULT indicating the result of previous operations (If SUCCEEDED(hrPrev) equals false, no operation is executed.) *)
	END_VAR

END_FUNCTION

// Functions/Container Statistics/F_VN_MinElementElementwise/F_VN_MinElementElementwise_LREAL

	{attribute 'TcIecLibraryType'}
	{attribute 'external_name' := 'F_VN_MinElementElementwise_LREAL_GUID_5A54C991_918C_B0AC_6726_7AB152DED603'}
	(* Gets the element wise minimum container element. *)
	FUNCTION F_VN_MinElementElementwise_LREAL : HRESULT
	VAR_INPUT
		ipContainer	:	ITcVnContainer;	(* Source container *)
	END_VAR
	VAR_IN_OUT
		fMin	:	LREAL;	(* Returns the requested element *)
	END_VAR
	VAR_INPUT
		hrPrev	:	HRESULT;	(* HRESULT indicating the result of previous operations (If SUCCEEDED(hrPrev) equals false, no operation is executed.) *)
	END_VAR

END_FUNCTION

// Functions/Container Statistics/F_VN_MinElementElementwise/F_VN_MinElementElementwise_REAL

	{attribute 'TcIecLibraryType'}
	{attribute 'external_name' := 'F_VN_MinElementElementwise_REAL_GUID_DE874430_ECF1_BF3D_5283_4E5BB53B780F'}
	(* Gets the element wise minimum container element. *)
	FUNCTION F_VN_MinElementElementwise_REAL : HRESULT
	VAR_INPUT
		ipContainer	:	ITcVnContainer;	(* Source container *)
	END_VAR
	VAR_IN_OUT
		fMin	:	REAL;	(* Returns the requested element *)
	END_VAR
	VAR_INPUT
		hrPrev	:	HRESULT;	(* HRESULT indicating the result of previous operations (If SUCCEEDED(hrPrev) equals false, no operation is executed.) *)
	END_VAR

END_FUNCTION

// Functions/Container Statistics/F_VN_MinElementElementwise/F_VN_MinElementElementwise_SINT

	{attribute 'TcIecLibraryType'}
	{attribute 'external_name' := 'F_VN_MinElementElementwise_SINT_GUID_B58CE3FD_A4E0_BB64_6957_C6CD3B3EB9A8'}
	(* Gets the element wise minimum container element. *)
	FUNCTION F_VN_MinElementElementwise_SINT : HRESULT
	VAR_INPUT
		ipContainer	:	ITcVnContainer;	(* Source container *)
	END_VAR
	VAR_IN_OUT
		nMin	:	SINT;	(* Returns the requested element *)
	END_VAR
	VAR_INPUT
		hrPrev	:	HRESULT;	(* HRESULT indicating the result of previous operations (If SUCCEEDED(hrPrev) equals false, no operation is executed.) *)
	END_VAR

END_FUNCTION

// Functions/Container Statistics/F_VN_MinElementElementwise/F_VN_MinElementElementwise_TcVnPoint2_DINT

	{attribute 'TcIecLibraryType'}
	{attribute 'external_name' := 'F_VN_MinElementElementwise_TcVnPoint2_DINT_GUID_95480FA3_5C50_BAFE_6E16_372142505BB2'}
	(* Gets the element wise minimum container element. *)
	FUNCTION F_VN_MinElementElementwise_TcVnPoint2_DINT : HRESULT
	VAR_INPUT
		ipContainer	:	ITcVnContainer;	(* Source container *)
	END_VAR
	VAR_IN_OUT
		aMin	:	TcVnPoint2_DINT;	(* Returns the requested element *)
	END_VAR
	VAR_INPUT
		hrPrev	:	HRESULT;	(* HRESULT indicating the result of previous operations (If SUCCEEDED(hrPrev) equals false, no operation is executed.) *)
	END_VAR

END_FUNCTION

// Functions/Container Statistics/F_VN_MinElementElementwise/F_VN_MinElementElementwise_TcVnPoint2_LREAL

	{attribute 'TcIecLibraryType'}
	{attribute 'external_name' := 'F_VN_MinElementElementwise_TcVnPoint2_LREAL_GUID_017D2D04_1941_BC59_50FF_283921CB7A72'}
	(* Gets the element wise minimum container element. *)
	FUNCTION F_VN_MinElementElementwise_TcVnPoint2_LREAL : HRESULT
	VAR_INPUT
		ipContainer	:	ITcVnContainer;	(* Source container *)
	END_VAR
	VAR_IN_OUT
		aMin	:	TcVnPoint2_LREAL;	(* Returns the requested element *)
	END_VAR
	VAR_INPUT
		hrPrev	:	HRESULT;	(* HRESULT indicating the result of previous operations (If SUCCEEDED(hrPrev) equals false, no operation is executed.) *)
	END_VAR

END_FUNCTION

// Functions/Container Statistics/F_VN_MinElementElementwise/F_VN_MinElementElementwise_TcVnPoint2_REAL

	{attribute 'TcIecLibraryType'}
	{attribute 'external_name' := 'F_VN_MinElementElementwise_TcVnPoint2_REAL_GUID_E147F811_4793_BB26_7EE1_51183C9B15D7'}
	(* Gets the element wise minimum container element. *)
	FUNCTION F_VN_MinElementElementwise_TcVnPoint2_REAL : HRESULT
	VAR_INPUT
		ipContainer	:	ITcVnContainer;	(* Source container *)
	END_VAR
	VAR_IN_OUT
		aMin	:	TcVnPoint2_REAL;	(* Returns the requested element *)
	END_VAR
	VAR_INPUT
		hrPrev	:	HRESULT;	(* HRESULT indicating the result of previous operations (If SUCCEEDED(hrPrev) equals false, no operation is executed.) *)
	END_VAR

END_FUNCTION

// Functions/Container Statistics/F_VN_MinElementElementwise/F_VN_MinElementElementwise_TcVnPoint3_LREAL

	{attribute 'TcIecLibraryType'}
	{attribute 'external_name' := 'F_VN_MinElementElementwise_TcVnPoint3_LREAL_GUID_2BAA822F_F1B6_B34E_6758_7FF701C9CC1D'}
	(* Gets the element wise minimum container element. *)
	FUNCTION F_VN_MinElementElementwise_TcVnPoint3_LREAL : HRESULT
	VAR_INPUT
		ipContainer	:	ITcVnContainer;	(* Source container *)
	END_VAR
	VAR_IN_OUT
		aMin	:	TcVnPoint3_LREAL;	(* Returns the requested element *)
	END_VAR
	VAR_INPUT
		hrPrev	:	HRESULT;	(* HRESULT indicating the result of previous operations (If SUCCEEDED(hrPrev) equals false, no operation is executed.) *)
	END_VAR

END_FUNCTION

// Functions/Container Statistics/F_VN_MinElementElementwise/F_VN_MinElementElementwise_TcVnPoint3_REAL

	{attribute 'TcIecLibraryType'}
	{attribute 'external_name' := 'F_VN_MinElementElementwise_TcVnPoint3_REAL_GUID_8DEFC356_AADF_BD8E_571D_EBBEB2E096F2'}
	(* Gets the element wise minimum container element. *)
	FUNCTION F_VN_MinElementElementwise_TcVnPoint3_REAL : HRESULT
	VAR_INPUT
		ipContainer	:	ITcVnContainer;	(* Source container *)
	END_VAR
	VAR_IN_OUT
		aMin	:	TcVnPoint3_REAL;	(* Returns the requested element *)
	END_VAR
	VAR_INPUT
		hrPrev	:	HRESULT;	(* HRESULT indicating the result of previous operations (If SUCCEEDED(hrPrev) equals false, no operation is executed.) *)
	END_VAR

END_FUNCTION

// Functions/Container Statistics/F_VN_MinElementElementwise/F_VN_MinElementElementwise_TcVnVector2_DINT

	{attribute 'TcIecLibraryType'}
	{attribute 'external_name' := 'F_VN_MinElementElementwise_TcVnVector2_DINT_GUID_D1716A90_334B_B087_74CF_F8EC8057490B'}
	(* Gets the element wise minimum container element. *)
	FUNCTION F_VN_MinElementElementwise_TcVnVector2_DINT : HRESULT
	VAR_INPUT
		ipContainer	:	ITcVnContainer;	(* Source container *)
	END_VAR
	VAR_IN_OUT
		aMin	:	TcVnVector2_DINT;	(* Returns the requested element *)
	END_VAR
	VAR_INPUT
		hrPrev	:	HRESULT;	(* HRESULT indicating the result of previous operations (If SUCCEEDED(hrPrev) equals false, no operation is executed.) *)
	END_VAR

END_FUNCTION

// Functions/Container Statistics/F_VN_MinElementElementwise/F_VN_MinElementElementwise_TcVnVector2_INT

	{attribute 'TcIecLibraryType'}
	{attribute 'external_name' := 'F_VN_MinElementElementwise_TcVnVector2_INT_GUID_CA1F7452_FEC6_B0A0_7566_6622B30AF87C'}
	(* Gets the element wise minimum container element. *)
	FUNCTION F_VN_MinElementElementwise_TcVnVector2_INT : HRESULT
	VAR_INPUT
		ipContainer	:	ITcVnContainer;	(* Source container *)
	END_VAR
	VAR_IN_OUT
		aMin	:	TcVnVector2_INT;	(* Returns the requested element *)
	END_VAR
	VAR_INPUT
		hrPrev	:	HRESULT;	(* HRESULT indicating the result of previous operations (If SUCCEEDED(hrPrev) equals false, no operation is executed.) *)
	END_VAR

END_FUNCTION

// Functions/Container Statistics/F_VN_MinElementElementwise/F_VN_MinElementElementwise_TcVnVector2_REAL

	{attribute 'TcIecLibraryType'}
	{attribute 'external_name' := 'F_VN_MinElementElementwise_TcVnVector2_REAL_GUID_1EAD29F1_DA5A_BA18_6D43_10367ABEF6D1'}
	(* Gets the element wise minimum container element. *)
	FUNCTION F_VN_MinElementElementwise_TcVnVector2_REAL : HRESULT
	VAR_INPUT
		ipContainer	:	ITcVnContainer;	(* Source container *)
	END_VAR
	VAR_IN_OUT
		aMin	:	TcVnVector2_REAL;	(* Returns the requested element *)
	END_VAR
	VAR_INPUT
		hrPrev	:	HRESULT;	(* HRESULT indicating the result of previous operations (If SUCCEEDED(hrPrev) equals false, no operation is executed.) *)
	END_VAR

END_FUNCTION

// Functions/Container Statistics/F_VN_MinElementElementwise/F_VN_MinElementElementwise_TcVnVector2_SINT

	{attribute 'TcIecLibraryType'}
	{attribute 'external_name' := 'F_VN_MinElementElementwise_TcVnVector2_SINT_GUID_DE4C7818_97E6_BF6C_5F55_F4EDC5FD5A58'}
	(* Gets the element wise minimum container element. *)
	FUNCTION F_VN_MinElementElementwise_TcVnVector2_SINT : HRESULT
	VAR_INPUT
		ipContainer	:	ITcVnContainer;	(* Source container *)
	END_VAR
	VAR_IN_OUT
		aMin	:	TcVnVector2_SINT;	(* Returns the requested element *)
	END_VAR
	VAR_INPUT
		hrPrev	:	HRESULT;	(* HRESULT indicating the result of previous operations (If SUCCEEDED(hrPrev) equals false, no operation is executed.) *)
	END_VAR

END_FUNCTION

// Functions/Container Statistics/F_VN_MinElementElementwise/F_VN_MinElementElementwise_TcVnVector2_UINT

	{attribute 'TcIecLibraryType'}
	{attribute 'external_name' := 'F_VN_MinElementElementwise_TcVnVector2_UINT_GUID_195C525C_ED89_BFAB_4A25_A79E6F132616'}
	(* Gets the element wise minimum container element. *)
	FUNCTION F_VN_MinElementElementwise_TcVnVector2_UINT : HRESULT
	VAR_INPUT
		ipContainer	:	ITcVnContainer;	(* Source container *)
	END_VAR
	VAR_IN_OUT
		aMin	:	TcVnVector2_UINT;	(* Returns the requested element *)
	END_VAR
	VAR_INPUT
		hrPrev	:	HRESULT;	(* HRESULT indicating the result of previous operations (If SUCCEEDED(hrPrev) equals false, no operation is executed.) *)
	END_VAR

END_FUNCTION

// Functions/Container Statistics/F_VN_MinElementElementwise/F_VN_MinElementElementwise_TcVnVector2_USINT

	{attribute 'TcIecLibraryType'}
	{attribute 'external_name' := 'F_VN_MinElementElementwise_TcVnVector2_USINT_GUID_4F4511EA_D31C_BCF7_4421_E65101E8EAC8'}
	(* Gets the element wise minimum container element. *)
	FUNCTION F_VN_MinElementElementwise_TcVnVector2_USINT : HRESULT
	VAR_INPUT
		ipContainer	:	ITcVnContainer;	(* Source container *)
	END_VAR
	VAR_IN_OUT
		aMin	:	TcVnVector2_USINT;	(* Returns the requested element *)
	END_VAR
	VAR_INPUT
		hrPrev	:	HRESULT;	(* HRESULT indicating the result of previous operations (If SUCCEEDED(hrPrev) equals false, no operation is executed.) *)
	END_VAR

END_FUNCTION

// Functions/Container Statistics/F_VN_MinElementElementwise/F_VN_MinElementElementwise_TcVnVector3_INT

	{attribute 'TcIecLibraryType'}
	{attribute 'external_name' := 'F_VN_MinElementElementwise_TcVnVector3_INT_GUID_9BBE78C6_23A9_B67A_54F6_6EFCF65A6B43'}
	(* Gets the element wise minimum container element. *)
	FUNCTION F_VN_MinElementElementwise_TcVnVector3_INT : HRESULT
	VAR_INPUT
		ipContainer	:	ITcVnContainer;	(* Source container *)
	END_VAR
	VAR_IN_OUT
		aMin	:	TcVnVector3_INT;	(* Returns the requested element *)
	END_VAR
	VAR_INPUT
		hrPrev	:	HRESULT;	(* HRESULT indicating the result of previous operations (If SUCCEEDED(hrPrev) equals false, no operation is executed.) *)
	END_VAR

END_FUNCTION

// Functions/Container Statistics/F_VN_MinElementElementwise/F_VN_MinElementElementwise_TcVnVector3_REAL

	{attribute 'TcIecLibraryType'}
	{attribute 'external_name' := 'F_VN_MinElementElementwise_TcVnVector3_REAL_GUID_577DF9B5_4D31_BE5A_71AA_C3D2358D4FA4'}
	(* Gets the element wise minimum container element. *)
	FUNCTION F_VN_MinElementElementwise_TcVnVector3_REAL : HRESULT
	VAR_INPUT
		ipContainer	:	ITcVnContainer;	(* Source container *)
	END_VAR
	VAR_IN_OUT
		aMin	:	TcVnVector3_REAL;	(* Returns the requested element *)
	END_VAR
	VAR_INPUT
		hrPrev	:	HRESULT;	(* HRESULT indicating the result of previous operations (If SUCCEEDED(hrPrev) equals false, no operation is executed.) *)
	END_VAR

END_FUNCTION

// Functions/Container Statistics/F_VN_MinElementElementwise/F_VN_MinElementElementwise_TcVnVector3_SINT

	{attribute 'TcIecLibraryType'}
	{attribute 'external_name' := 'F_VN_MinElementElementwise_TcVnVector3_SINT_GUID_FB3ADB12_1F37_B2CA_4BC2_75B2EB2A831F'}
	(* Gets the element wise minimum container element. *)
	FUNCTION F_VN_MinElementElementwise_TcVnVector3_SINT : HRESULT
	VAR_INPUT
		ipContainer	:	ITcVnContainer;	(* Source container *)
	END_VAR
	VAR_IN_OUT
		aMin	:	TcVnVector3_SINT;	(* Returns the requested element *)
	END_VAR
	VAR_INPUT
		hrPrev	:	HRESULT;	(* HRESULT indicating the result of previous operations (If SUCCEEDED(hrPrev) equals false, no operation is executed.) *)
	END_VAR

END_FUNCTION

// Functions/Container Statistics/F_VN_MinElementElementwise/F_VN_MinElementElementwise_TcVnVector3_UINT

	{attribute 'TcIecLibraryType'}
	{attribute 'external_name' := 'F_VN_MinElementElementwise_TcVnVector3_UINT_GUID_A92AD152_DBFA_B8D7_53F7_30D3A9572EB0'}
	(* Gets the element wise minimum container element. *)
	FUNCTION F_VN_MinElementElementwise_TcVnVector3_UINT : HRESULT
	VAR_INPUT
		ipContainer	:	ITcVnContainer;	(* Source container *)
	END_VAR
	VAR_IN_OUT
		aMin	:	TcVnVector3_UINT;	(* Returns the requested element *)
	END_VAR
	VAR_INPUT
		hrPrev	:	HRESULT;	(* HRESULT indicating the result of previous operations (If SUCCEEDED(hrPrev) equals false, no operation is executed.) *)
	END_VAR

END_FUNCTION

// Functions/Container Statistics/F_VN_MinElementElementwise/F_VN_MinElementElementwise_TcVnVector3_USINT

	{attribute 'TcIecLibraryType'}
	{attribute 'external_name' := 'F_VN_MinElementElementwise_TcVnVector3_USINT_GUID_F7669910_CA88_B516_5183_7D209BF2C823'}
	(* Gets the element wise minimum container element. *)
	FUNCTION F_VN_MinElementElementwise_TcVnVector3_USINT : HRESULT
	VAR_INPUT
		ipContainer	:	ITcVnContainer;	(* Source container *)
	END_VAR
	VAR_IN_OUT
		aMin	:	TcVnVector3_USINT;	(* Returns the requested element *)
	END_VAR
	VAR_INPUT
		hrPrev	:	HRESULT;	(* HRESULT indicating the result of previous operations (If SUCCEEDED(hrPrev) equals false, no operation is executed.) *)
	END_VAR

END_FUNCTION

// Functions/Container Statistics/F_VN_MinElementElementwise/F_VN_MinElementElementwise_TcVnVector4_DINT

	{attribute 'TcIecLibraryType'}
	{attribute 'external_name' := 'F_VN_MinElementElementwise_TcVnVector4_DINT_GUID_D1CE795E_3BAF_B873_7CE3_48E16E25F696'}
	(* Gets the element wise minimum container element. *)
	FUNCTION F_VN_MinElementElementwise_TcVnVector4_DINT : HRESULT
	VAR_INPUT
		ipContainer	:	ITcVnContainer;	(* Source container *)
	END_VAR
	VAR_IN_OUT
		aMin	:	TcVnVector4_DINT;	(* Returns the requested element *)
	END_VAR
	VAR_INPUT
		hrPrev	:	HRESULT;	(* HRESULT indicating the result of previous operations (If SUCCEEDED(hrPrev) equals false, no operation is executed.) *)
	END_VAR

END_FUNCTION

// Functions/Container Statistics/F_VN_MinElementElementwise/F_VN_MinElementElementwise_TcVnVector4_INT

	{attribute 'TcIecLibraryType'}
	{attribute 'external_name' := 'F_VN_MinElementElementwise_TcVnVector4_INT_GUID_6FEB6493_B7A8_B8FC_75BB_A73C2A65EFA5'}
	(* Gets the element wise minimum container element. *)
	FUNCTION F_VN_MinElementElementwise_TcVnVector4_INT : HRESULT
	VAR_INPUT
		ipContainer	:	ITcVnContainer;	(* Source container *)
	END_VAR
	VAR_IN_OUT
		aMin	:	TcVnVector4_INT;	(* Returns the requested element *)
	END_VAR
	VAR_INPUT
		hrPrev	:	HRESULT;	(* HRESULT indicating the result of previous operations (If SUCCEEDED(hrPrev) equals false, no operation is executed.) *)
	END_VAR

END_FUNCTION

// Functions/Container Statistics/F_VN_MinElementElementwise/F_VN_MinElementElementwise_TcVnVector4_LREAL

	{attribute 'TcIecLibraryType'}
	{attribute 'external_name' := 'F_VN_MinElementElementwise_TcVnVector4_LREAL_GUID_5705740D_3ED9_BFBD_5716_3C31D7525AC1'}
	(* Gets the element wise minimum container element. *)
	FUNCTION F_VN_MinElementElementwise_TcVnVector4_LREAL : HRESULT
	VAR_INPUT
		ipContainer	:	ITcVnContainer;	(* Source container *)
	END_VAR
	VAR_IN_OUT
		aMin	:	TcVnVector4_LREAL;	(* Returns the requested element *)
	END_VAR
	VAR_INPUT
		hrPrev	:	HRESULT;	(* HRESULT indicating the result of previous operations (If SUCCEEDED(hrPrev) equals false, no operation is executed.) *)
	END_VAR

END_FUNCTION

// Functions/Container Statistics/F_VN_MinElementElementwise/F_VN_MinElementElementwise_TcVnVector4_SINT

	{attribute 'TcIecLibraryType'}
	{attribute 'external_name' := 'F_VN_MinElementElementwise_TcVnVector4_SINT_GUID_889E25AE_6E2D_B31D_74D3_982003F4CE0D'}
	(* Gets the element wise minimum container element. *)
	FUNCTION F_VN_MinElementElementwise_TcVnVector4_SINT : HRESULT
	VAR_INPUT
		ipContainer	:	ITcVnContainer;	(* Source container *)
	END_VAR
	VAR_IN_OUT
		aMin	:	TcVnVector4_SINT;	(* Returns the requested element *)
	END_VAR
	VAR_INPUT
		hrPrev	:	HRESULT;	(* HRESULT indicating the result of previous operations (If SUCCEEDED(hrPrev) equals false, no operation is executed.) *)
	END_VAR

END_FUNCTION

// Functions/Container Statistics/F_VN_MinElementElementwise/F_VN_MinElementElementwise_TcVnVector4_UINT

	{attribute 'TcIecLibraryType'}
	{attribute 'external_name' := 'F_VN_MinElementElementwise_TcVnVector4_UINT_GUID_47455897_585D_B050_495B_84CBA1F0D496'}
	(* Gets the element wise minimum container element. *)
	FUNCTION F_VN_MinElementElementwise_TcVnVector4_UINT : HRESULT
	VAR_INPUT
		ipContainer	:	ITcVnContainer;	(* Source container *)
	END_VAR
	VAR_IN_OUT
		aMin	:	TcVnVector4_UINT;	(* Returns the requested element *)
	END_VAR
	VAR_INPUT
		hrPrev	:	HRESULT;	(* HRESULT indicating the result of previous operations (If SUCCEEDED(hrPrev) equals false, no operation is executed.) *)
	END_VAR

END_FUNCTION

// Functions/Container Statistics/F_VN_MinElementElementwise/F_VN_MinElementElementwise_TcVnVector4_USINT

	{attribute 'TcIecLibraryType'}
	{attribute 'external_name' := 'F_VN_MinElementElementwise_TcVnVector4_USINT_GUID_E05F7B5F_2AEE_B843_6566_830535EA0543'}
	(* Gets the element wise minimum container element. *)
	FUNCTION F_VN_MinElementElementwise_TcVnVector4_USINT : HRESULT
	VAR_INPUT
		ipContainer	:	ITcVnContainer;	(* Source container *)
	END_VAR
	VAR_IN_OUT
		aMin	:	TcVnVector4_USINT;	(* Returns the requested element *)
	END_VAR
	VAR_INPUT
		hrPrev	:	HRESULT;	(* HRESULT indicating the result of previous operations (If SUCCEEDED(hrPrev) equals false, no operation is executed.) *)
	END_VAR

END_FUNCTION

// Functions/Container Statistics/F_VN_MinElementElementwise/F_VN_MinElementElementwise_UDINT

	{attribute 'TcIecLibraryType'}
	{attribute 'external_name' := 'F_VN_MinElementElementwise_UDINT_GUID_EB577D13_0852_BF0C_54E8_BC721109721D'}
	(* Gets the element wise minimum container element. *)
	FUNCTION F_VN_MinElementElementwise_UDINT : HRESULT
	VAR_INPUT
		ipContainer	:	ITcVnContainer;	(* Source container *)
	END_VAR
	VAR_IN_OUT
		nMin	:	UDINT;	(* Returns the requested element *)
	END_VAR
	VAR_INPUT
		hrPrev	:	HRESULT;	(* HRESULT indicating the result of previous operations (If SUCCEEDED(hrPrev) equals false, no operation is executed.) *)
	END_VAR

END_FUNCTION

// Functions/Container Statistics/F_VN_MinElementElementwise/F_VN_MinElementElementwise_UINT

	{attribute 'TcIecLibraryType'}
	{attribute 'external_name' := 'F_VN_MinElementElementwise_UINT_GUID_EA902095_0BC1_B543_63F5_57B77E38950D'}
	(* Gets the element wise minimum container element. *)
	FUNCTION F_VN_MinElementElementwise_UINT : HRESULT
	VAR_INPUT
		ipContainer	:	ITcVnContainer;	(* Source container *)
	END_VAR
	VAR_IN_OUT
		nMin	:	UINT;	(* Returns the requested element *)
	END_VAR
	VAR_INPUT
		hrPrev	:	HRESULT;	(* HRESULT indicating the result of previous operations (If SUCCEEDED(hrPrev) equals false, no operation is executed.) *)
	END_VAR

END_FUNCTION

// Functions/Container Statistics/F_VN_MinElementElementwise/F_VN_MinElementElementwise_ULINT

	{attribute 'TcIecLibraryType'}
	{attribute 'external_name' := 'F_VN_MinElementElementwise_ULINT_GUID_7BBE014E_3E13_B1BE_5C2C_440348C8244C'}
	(* Gets the element wise minimum container element. *)
	FUNCTION F_VN_MinElementElementwise_ULINT : HRESULT
	VAR_INPUT
		ipContainer	:	ITcVnContainer;	(* Source container *)
	END_VAR
	VAR_IN_OUT
		nMin	:	ULINT;	(* Returns the requested element *)
	END_VAR
	VAR_INPUT
		hrPrev	:	HRESULT;	(* HRESULT indicating the result of previous operations (If SUCCEEDED(hrPrev) equals false, no operation is executed.) *)
	END_VAR

END_FUNCTION

// Functions/Container Statistics/F_VN_MinElementElementwise/F_VN_MinElementElementwise_USINT

	{attribute 'TcIecLibraryType'}
	{attribute 'external_name' := 'F_VN_MinElementElementwise_USINT_GUID_ABB08848_8A93_BDF0_62BA_7A44177822DA'}
	(* Gets the element wise minimum container element. *)
	FUNCTION F_VN_MinElementElementwise_USINT : HRESULT
	VAR_INPUT
		ipContainer	:	ITcVnContainer;	(* Source container *)
	END_VAR
	VAR_IN_OUT
		nMin	:	USINT;	(* Returns the requested element *)
	END_VAR
	VAR_INPUT
		hrPrev	:	HRESULT;	(* HRESULT indicating the result of previous operations (If SUCCEEDED(hrPrev) equals false, no operation is executed.) *)
	END_VAR

END_FUNCTION
